// TwinCAT 3 PLC project PLC1
// ProgramVersion: 3.1.4026.27
// libraries:
//   Tc2_Standard, * (Beckhoff Automation GmbH)
//   Tc2_System, * (Beckhoff Automation GmbH)
//   Tc2_Utilities, * (Beckhoff Automation GmbH)
//   XPlanarApplication, * (Beckhoff Automation LLC)
// project tree:
//   DemoStep/ E_DemoStep.TcDUT, I_BothMovers.TcIO, I_Errorable.TcIO, I_SingleMover.TcIO, I_XplanarTable.TcIO, I_DemoStep.TcIO
//   DemoStep/Steps/ DetectXplanarMovers.TcPOU, LiftMove.TcPOU, SimpleDisableWithRotSwAndEstop.TcPOU, SimpleDisableWithPB.TcPOU, TiltMove.TcPOU, SpinMove.TcPOU, MoveAroundPerimeter.TcPOU, JoinAllClosestTracks.TcPOU, MoveAroundInSequence.TcPOU, OscillateRotateMove.TcPOU, RecoverMoveToAnyPos.TcPOU, FlyByMove.TcPOU, MoveToCenters.TcPOU, SameTrackMove.TcPOU, LeaveAllTracks.TcPOU, SimpleSort2Movers.TcPOU, SquareUpMovers.TcPOU, WaitForRotSw.TcPOU, InitStep.TcPOU, WaitForPB.TcPOU
//   DUTs/EStop/ E_EStop.TcDUT, ST_EstopIO.TcDUT, U_Estop.TcDUT
//   DUTs/ E_ButtonColors.TcDUT, E_UsbLicenseDongleSate.TcDUT, ST_Point.TcDUT (not stored)
//   DUTs/SelectorSwitch/ E_SelectorSwitchPos.TcDUT, ST_SelectorSwitchIO.TcDUT, U_SelectorSwitch.TcDUT
//   GVLs/ CoorPoint2Tile.TcGVL, Defaults.TcGVL
//   / PlcTask.TcTTO
//   POUs/ FB_PushButton.TcPOU, FB_ToggleButton.TcPOU, F_FindCorrectOpposingCornerPosition.TcPOU, F_FindOpposingRotationPosition.TcPOU, F_SetAllMoversMovement.TcPOU (not stored), F_SetAllMoversRotation.TcPOU (not stored), I_DemoSystem.TcIO, MAIN.TcPOU
// real-time tasks:
//   TASK PlcTask: cycle T#1ms, priority 20, ADS port 350
//   TASK Job Task: cycle default, priority 32
//   TASK XPlanar Task_3: cycle T#250us, priority 1, ADS port 351
//   TASK MC-Task (MET): cycle T#2ms, priority 2, ADS port 352
//   TASK MC-Task (MPT): cycle T#10ms, priority 3, ADS port 353
// I/O:
//   DEVICE XPlanar, AmsNetId 0.0.0.0.4.1
//     Term 1 (APS4322-7000) [APS4322-7000 Drive]
//       Term 2 (APS4322-5000) [APS4322-5000 Feedback]
//     Term 3 (APS4322-7000) [APS4322-7000 Drive]
//       Term 4 (APS4322-5000) [APS4322-5000 Feedback]
//   DEVICE IO (EtherCAT), AmsNetId 0.0.0.0.2.1
//     EtherCAT PS (PS2001-2410) [PS2001-2410-1001 Power supply (24V, 10A, 1-phase)]
//     IoLink PushButtons (EP6224-0002) [EP6224-0002 (IO Link Master)]
//       modules: Module 1 (DeviceState Inputs Device), Module 2 (DeviceState Inputs), Port1 (CANEO series10 Hygienic), Port2 (CANEO series10 Hygienic), Port3 (CANEO series10 Hygienic), Module 6 (empty), Module 7 (Digital Inputs)
//     DIO Box (RS and ESTOP) (EP2316-0003) [EP2316-0003 8 Ch. Dig. In, 10µs, 8Ch. Dig. Out 24V, 0,5A, Diagnostic, 10-Pole Plug Connector] (disabled)
//   DEVICE USB
//     Box 2 (C9900-L100 License-Key-USB-Stick)
// variable links:
//   PLC1/PLC1 Instance <-> IO (EtherCAT)
//     PlcTask Inputs/MAIN.IODeviceState <-> Inputs/DevState
//   PLC1/PLC1 Instance <-> USB/Box 2 (C9900-L100 License-Key-USB-Stick)
//     PlcTask Inputs/MAIN.LicUsbState <-> BoxInfo/BoxState
//   PLC1/PLC1 Instance <-> XPlanar
//     PlcTask Inputs/MAIN.XPlanarDeviceState <-> Inputs/DevState
//   PLC1/PLC1 Instance <-> XPlanar MC Project/Axes/Mover4220_1
//     PlcTask Inputs/MAIN.Mover1._Mover.MCTOPLC/ACT <-> McToPlc/ACT
//     PlcTask Inputs/MAIN.Mover1._Mover.MCTOPLC/COORDMODE <-> McToPlc/COORDMODE
//     PlcTask Inputs/MAIN.Mover1._Mover.MCTOPLC/SET <-> McToPlc/SET
//     PlcTask Inputs/MAIN.Mover1._Mover.MCTOPLC/SETONTRACK <-> McToPlc/SETONTRACK
//     PlcTask Inputs/MAIN.Mover1._Mover.MCTOPLC/STD <-> McToPlc/STD
//     PlcTask Outputs/MAIN.Mover1._Mover.PLCTOMC/STD <-> PlcToMc/STD
//   PLC1/PLC1 Instance <-> XPlanar MC Project/Axes/Mover4220_2
//     PlcTask Inputs/MAIN.Mover2._Mover.MCTOPLC/ACT <-> McToPlc/ACT
//     PlcTask Inputs/MAIN.Mover2._Mover.MCTOPLC/COORDMODE <-> McToPlc/COORDMODE
//     PlcTask Inputs/MAIN.Mover2._Mover.MCTOPLC/SET <-> McToPlc/SET
//     PlcTask Inputs/MAIN.Mover2._Mover.MCTOPLC/SETONTRACK <-> McToPlc/SETONTRACK
//     PlcTask Inputs/MAIN.Mover2._Mover.MCTOPLC/STD <-> McToPlc/STD
//     PlcTask Outputs/MAIN.Mover2._Mover.PLCTOMC/STD <-> PlcToMc/STD
//   PLC1/PLC1 Instance <-> XPlanar MC Project/Groups/Environment
//     PlcTask Inputs/XPlanar.Environment.MCTOPLC_STD <-> McToPlc/STD
//   PLC1/PLC1 Instance <-> XPlanar MC Project/Groups/Track_Fig8
//     PlcTask Inputs/MAIN.Track1._Track.MCTOPLC_STD <-> McToPlc/STD
//   PLC1/PLC1 Instance <-> XPlanar MC Project/Groups/XPlanar
//     PlcTask Inputs/XPlanar.Group.MCTOPLC_STD <-> McToPlc/STD
//   TcCOM Objects/XPlanar <-> XPlanar/Term 1 (APS4322-7000)
//     Part1/APS4322_P1_2/Data Pointer/DCurrentSetPoints[0] <-> APS Outputs/Current D 0X0
//     Part1/APS4322_P1_2/Data Pointer/DCurrentSetPoints[12] <-> APS Outputs/Current D 2X0
//     Part1/APS4322_P1_2/Data Pointer/DCurrentSetPoints[13] <-> APS Outputs/Current D 2X1
//     Part1/APS4322_P1_2/Data Pointer/DCurrentSetPoints[14] <-> APS Outputs/Current D 2X2
//     Part1/APS4322_P1_2/Data Pointer/DCurrentSetPoints[18] <-> APS Outputs/Current D 3X0
//     Part1/APS4322_P1_2/Data Pointer/DCurrentSetPoints[19] <-> APS Outputs/Current D 3X1
//     Part1/APS4322_P1_2/Data Pointer/DCurrentSetPoints[1] <-> APS Outputs/Current D 0X1
//     Part1/APS4322_P1_2/Data Pointer/DCurrentSetPoints[20] <-> APS Outputs/Current D 3X2
//     Part1/APS4322_P1_2/Data Pointer/DCurrentSetPoints[2] <-> APS Outputs/Current D 0X2
//     Part1/APS4322_P1_2/Data Pointer/DCurrentSetPoints[6] <-> APS Outputs/Current D 1X0
//     Part1/APS4322_P1_2/Data Pointer/DCurrentSetPoints[7] <-> APS Outputs/Current D 1X1
//     Part1/APS4322_P1_2/Data Pointer/DCurrentSetPoints[8] <-> APS Outputs/Current D 1X2
//     Part1/APS4322_P1_2/Data Pointer/DCurrentSetPoints[10] <-> APS Outputs/Current D 1Y1
//     Part1/APS4322_P1_2/Data Pointer/DCurrentSetPoints[11] <-> APS Outputs/Current D 1Y2
//     Part1/APS4322_P1_2/Data Pointer/DCurrentSetPoints[15] <-> APS Outputs/Current D 2Y0
//     Part1/APS4322_P1_2/Data Pointer/DCurrentSetPoints[16] <-> APS Outputs/Current D 2Y1
//     Part1/APS4322_P1_2/Data Pointer/DCurrentSetPoints[17] <-> APS Outputs/Current D 2Y2
//     Part1/APS4322_P1_2/Data Pointer/DCurrentSetPoints[21] <-> APS Outputs/Current D 3Y0
//     Part1/APS4322_P1_2/Data Pointer/DCurrentSetPoints[22] <-> APS Outputs/Current D 3Y1
//     Part1/APS4322_P1_2/Data Pointer/DCurrentSetPoints[23] <-> APS Outputs/Current D 3Y2
//     Part1/APS4322_P1_2/Data Pointer/DCurrentSetPoints[3] <-> APS Outputs/Current D 0Y0
//     Part1/APS4322_P1_2/Data Pointer/DCurrentSetPoints[4] <-> APS Outputs/Current D 0Y1
//     Part1/APS4322_P1_2/Data Pointer/DCurrentSetPoints[5] <-> APS Outputs/Current D 0Y2
//     Part1/APS4322_P1_2/Data Pointer/DCurrentSetPoints[9] <-> APS Outputs/Current D 1Y0
//     Part1/APS4322_P1_2/Data Pointer/DcLinkVoltage <-> APS Diagdata/DC Link Voltage
//     Part1/APS4322_P1_2/Data Pointer/MoverCommControlWord <-> APS Comm Outputs/CommControlWord
//     Part1/APS4322_P1_2/Data Pointer/MoverCommDataIn[{0..3}] <-> APS Comm Inputs/Data {1..4}  (4 links)
//     Part1/APS4322_P1_2/Data Pointer/MoverCommDataOut <-> APS Comm Outputs/Data 1
//     Part1/APS4322_P1_2/Data Pointer/MoverCommStatusWord <-> APS Comm Inputs/CommStatusWord
//     Part1/APS4322_P1_2/Data Pointer/PhiSetPoints[0] <-> APS Outputs/PhiE 0X0
//     Part1/APS4322_P1_2/Data Pointer/PhiSetPoints[12] <-> APS Outputs/PhiE 2X0
//     Part1/APS4322_P1_2/Data Pointer/PhiSetPoints[13] <-> APS Outputs/PhiE 2X1
//     Part1/APS4322_P1_2/Data Pointer/PhiSetPoints[14] <-> APS Outputs/PhiE 2X2
//     Part1/APS4322_P1_2/Data Pointer/PhiSetPoints[18] <-> APS Outputs/PhiE 3X0
//     Part1/APS4322_P1_2/Data Pointer/PhiSetPoints[19] <-> APS Outputs/PhiE 3X1
//     Part1/APS4322_P1_2/Data Pointer/PhiSetPoints[1] <-> APS Outputs/PhiE 0X1
//     Part1/APS4322_P1_2/Data Pointer/PhiSetPoints[20] <-> APS Outputs/PhiE 3X2
//     Part1/APS4322_P1_2/Data Pointer/PhiSetPoints[2] <-> APS Outputs/PhiE 0X2
//     Part1/APS4322_P1_2/Data Pointer/PhiSetPoints[6] <-> APS Outputs/PhiE 1X0
//     Part1/APS4322_P1_2/Data Pointer/PhiSetPoints[7] <-> APS Outputs/PhiE 1X1
//     Part1/APS4322_P1_2/Data Pointer/PhiSetPoints[8] <-> APS Outputs/PhiE 1X2
//     Part1/APS4322_P1_2/Data Pointer/PhiSetPoints[10] <-> APS Outputs/PhiE 1Y1
//     Part1/APS4322_P1_2/Data Pointer/PhiSetPoints[11] <-> APS Outputs/PhiE 1Y2
//     Part1/APS4322_P1_2/Data Pointer/PhiSetPoints[15] <-> APS Outputs/PhiE 2Y0
//     Part1/APS4322_P1_2/Data Pointer/PhiSetPoints[16] <-> APS Outputs/PhiE 2Y1
//     Part1/APS4322_P1_2/Data Pointer/PhiSetPoints[17] <-> APS Outputs/PhiE 2Y2
//     Part1/APS4322_P1_2/Data Pointer/PhiSetPoints[21] <-> APS Outputs/PhiE 3Y0
//     Part1/APS4322_P1_2/Data Pointer/PhiSetPoints[22] <-> APS Outputs/PhiE 3Y1
//     Part1/APS4322_P1_2/Data Pointer/PhiSetPoints[23] <-> APS Outputs/PhiE 3Y2
//     Part1/APS4322_P1_2/Data Pointer/PhiSetPoints[3] <-> APS Outputs/PhiE 0Y0
//     Part1/APS4322_P1_2/Data Pointer/PhiSetPoints[4] <-> APS Outputs/PhiE 0Y1
//     Part1/APS4322_P1_2/Data Pointer/PhiSetPoints[5] <-> APS Outputs/PhiE 0Y2
//     Part1/APS4322_P1_2/Data Pointer/PhiSetPoints[9] <-> APS Outputs/PhiE 1Y0
//     Part1/APS4322_P1_2/Data Pointer/PowerSupplyCurrent <-> APS Diagdata/Power supply current
//     Part1/APS4322_P1_2/Data Pointer/PowerUnitControlWord <-> APS Outputs/ControlWord
//     Part1/APS4322_P1_2/Data Pointer/PowerUnitStatusWord <-> APS Inputs/StatusWord
//     Part1/APS4322_P1_2/Data Pointer/QCurrentSetPoints[0] <-> APS Outputs/Current Q 0X0
//     Part1/APS4322_P1_2/Data Pointer/QCurrentSetPoints[12] <-> APS Outputs/Current Q 2X0
//     Part1/APS4322_P1_2/Data Pointer/QCurrentSetPoints[13] <-> APS Outputs/Current Q 2X1
//     Part1/APS4322_P1_2/Data Pointer/QCurrentSetPoints[14] <-> APS Outputs/Current Q 2X2
//     Part1/APS4322_P1_2/Data Pointer/QCurrentSetPoints[18] <-> APS Outputs/Current Q 3X0
//     Part1/APS4322_P1_2/Data Pointer/QCurrentSetPoints[19] <-> APS Outputs/Current Q 3X1
//     Part1/APS4322_P1_2/Data Pointer/QCurrentSetPoints[1] <-> APS Outputs/Current Q 0X1
//     Part1/APS4322_P1_2/Data Pointer/QCurrentSetPoints[20] <-> APS Outputs/Current Q 3X2
//     Part1/APS4322_P1_2/Data Pointer/QCurrentSetPoints[2] <-> APS Outputs/Current Q 0X2
//     Part1/APS4322_P1_2/Data Pointer/QCurrentSetPoints[6] <-> APS Outputs/Current Q 1X0
//     Part1/APS4322_P1_2/Data Pointer/QCurrentSetPoints[7] <-> APS Outputs/Current Q 1X1
//     Part1/APS4322_P1_2/Data Pointer/QCurrentSetPoints[8] <-> APS Outputs/Current Q 1X2
//     Part1/APS4322_P1_2/Data Pointer/QCurrentSetPoints[10] <-> APS Outputs/Current Q 1Y1
//     Part1/APS4322_P1_2/Data Pointer/QCurrentSetPoints[11] <-> APS Outputs/Current Q 1Y2
//     Part1/APS4322_P1_2/Data Pointer/QCurrentSetPoints[15] <-> APS Outputs/Current Q 2Y0
//     Part1/APS4322_P1_2/Data Pointer/QCurrentSetPoints[16] <-> APS Outputs/Current Q 2Y1
//     Part1/APS4322_P1_2/Data Pointer/QCurrentSetPoints[17] <-> APS Outputs/Current Q 2Y2
//     Part1/APS4322_P1_2/Data Pointer/QCurrentSetPoints[21] <-> APS Outputs/Current Q 3Y0
//     Part1/APS4322_P1_2/Data Pointer/QCurrentSetPoints[22] <-> APS Outputs/Current Q 3Y1
//     Part1/APS4322_P1_2/Data Pointer/QCurrentSetPoints[23] <-> APS Outputs/Current Q 3Y2
//     Part1/APS4322_P1_2/Data Pointer/QCurrentSetPoints[3] <-> APS Outputs/Current Q 0Y0
//     Part1/APS4322_P1_2/Data Pointer/QCurrentSetPoints[4] <-> APS Outputs/Current Q 0Y1
//     Part1/APS4322_P1_2/Data Pointer/QCurrentSetPoints[5] <-> APS Outputs/Current Q 0Y2
//     Part1/APS4322_P1_2/Data Pointer/QCurrentSetPoints[9] <-> APS Outputs/Current Q 1Y0
//   TcCOM Objects/XPlanar <-> XPlanar/Term 1 (APS4322-7000)/Term 2 (APS4322-5000)
//     Part1/APS4322_P1_2/Data Pointer/FeedbackStatus <-> FB Inputs/Status
//     Part1/APS4322_P1_2/Data Pointer/HallSensorFieldsXYZ[{0..12 step 3}] <-> FB Inputs/A{0..8 step 2} X-Field  (5 links)
//     Part1/APS4322_P1_2/Data Pointer/HallSensorFieldsXYZ[{91..103 step 3}] <-> FB Inputs/G{0..8 step 2} Y-Field  (5 links)
//     Part1/APS4322_P1_2/Data Pointer/HallSensorFieldsXYZ[{92..104 step 3}] <-> FB Inputs/G{0..8 step 2} Z-Field  (5 links)
//     Part1/APS4322_P1_2/Data Pointer/HallSensorFieldsXYZ[{90..102 step 3}] <-> FB Inputs/G{0..8 step 2} X-Field  (5 links)
//     Part1/APS4322_P1_2/Data Pointer/HallSensorFieldsXYZ[{105..117 step 3}] <-> FB Inputs/H{1..9 step 2} X-Field  (5 links)
//     Part1/APS4322_P1_2/Data Pointer/HallSensorFieldsXYZ[{106..118 step 3}] <-> FB Inputs/H{1..9 step 2} Y-Field  (5 links)
//     Part1/APS4322_P1_2/Data Pointer/HallSensorFieldsXYZ[{107..119 step 3}] <-> FB Inputs/H{1..9 step 2} Z-Field  (5 links)
//     Part1/APS4322_P1_2/Data Pointer/HallSensorFieldsXYZ[{1..13 step 3}] <-> FB Inputs/A{0..8 step 2} Y-Field  (5 links)
//     Part1/APS4322_P1_2/Data Pointer/HallSensorFieldsXYZ[{2..14 step 3}] <-> FB Inputs/A{0..8 step 2} Z-Field  (5 links)
//     Part1/APS4322_P1_2/Data Pointer/HallSensorFieldsXYZ[{120..132 step 3}] <-> FB Inputs/I{0..8 step 2} X-Field  (5 links)
//     Part1/APS4322_P1_2/Data Pointer/HallSensorFieldsXYZ[{121..133 step 3}] <-> FB Inputs/I{0..8 step 2} Y-Field  (5 links)
//     Part1/APS4322_P1_2/Data Pointer/HallSensorFieldsXYZ[{122..134 step 3}] <-> FB Inputs/I{0..8 step 2} Z-Field  (5 links)
//     Part1/APS4322_P1_2/Data Pointer/HallSensorFieldsXYZ[{135..147 step 3}] <-> FB Inputs/J{1..9 step 2} X-Field  (5 links)
//     Part1/APS4322_P1_2/Data Pointer/HallSensorFieldsXYZ[{136..148 step 3}] <-> FB Inputs/J{1..9 step 2} Y-Field  (5 links)
//     Part1/APS4322_P1_2/Data Pointer/HallSensorFieldsXYZ[{137..149 step 3}] <-> FB Inputs/J{1..9 step 2} Z-Field  (5 links)
//     Part1/APS4322_P1_2/Data Pointer/HallSensorFieldsXYZ[{15..27 step 3}] <-> FB Inputs/B{1..9 step 2} X-Field  (5 links)
//     Part1/APS4322_P1_2/Data Pointer/HallSensorFieldsXYZ[{16..28 step 3}] <-> FB Inputs/B{1..9 step 2} Y-Field  (5 links)
//     Part1/APS4322_P1_2/Data Pointer/HallSensorFieldsXYZ[{17..29 step 3}] <-> FB Inputs/B{1..9 step 2} Z-Field  (5 links)
//     Part1/APS4322_P1_2/Data Pointer/HallSensorFieldsXYZ[{30..42 step 3}] <-> FB Inputs/C{0..8 step 2} X-Field  (5 links)
//     Part1/APS4322_P1_2/Data Pointer/HallSensorFieldsXYZ[{31..43 step 3}] <-> FB Inputs/C{0..8 step 2} Y-Field  (5 links)
//     Part1/APS4322_P1_2/Data Pointer/HallSensorFieldsXYZ[{32..44 step 3}] <-> FB Inputs/C{0..8 step 2} Z-Field  (5 links)
//     Part1/APS4322_P1_2/Data Pointer/HallSensorFieldsXYZ[{45..57 step 3}] <-> FB Inputs/D{1..9 step 2} X-Field  (5 links)
//     Part1/APS4322_P1_2/Data Pointer/HallSensorFieldsXYZ[{46..58 step 3}] <-> FB Inputs/D{1..9 step 2} Y-Field  (5 links)
//     Part1/APS4322_P1_2/Data Pointer/HallSensorFieldsXYZ[{47..59 step 3}] <-> FB Inputs/D{1..9 step 2} Z-Field  (5 links)
//     Part1/APS4322_P1_2/Data Pointer/HallSensorFieldsXYZ[{60..72 step 3}] <-> FB Inputs/E{0..8 step 2} X-Field  (5 links)
//     Part1/APS4322_P1_2/Data Pointer/HallSensorFieldsXYZ[{61..73 step 3}] <-> FB Inputs/E{0..8 step 2} Y-Field  (5 links)
//     Part1/APS4322_P1_2/Data Pointer/HallSensorFieldsXYZ[{62..74 step 3}] <-> FB Inputs/E{0..8 step 2} Z-Field  (5 links)
//     Part1/APS4322_P1_2/Data Pointer/HallSensorFieldsXYZ[{75..87 step 3}] <-> FB Inputs/F{1..9 step 2} X-Field  (5 links)
//     Part1/APS4322_P1_2/Data Pointer/HallSensorFieldsXYZ[{76..88 step 3}] <-> FB Inputs/F{1..9 step 2} Y-Field  (5 links)
//     Part1/APS4322_P1_2/Data Pointer/HallSensorFieldsXYZ[{77..89 step 3}] <-> FB Inputs/F{1..9 step 2} Z-Field  (5 links)
//   TcCOM Objects/XPlanar <-> XPlanar/Term 3 (APS4322-7000)
//     Part1/APS4322_P1_1/Data Pointer/DCurrentSetPoints[0] <-> APS Outputs/Current D 0X0
//     Part1/APS4322_P1_1/Data Pointer/DCurrentSetPoints[12] <-> APS Outputs/Current D 2X0
//     Part1/APS4322_P1_1/Data Pointer/DCurrentSetPoints[13] <-> APS Outputs/Current D 2X1
//     Part1/APS4322_P1_1/Data Pointer/DCurrentSetPoints[14] <-> APS Outputs/Current D 2X2
//     Part1/APS4322_P1_1/Data Pointer/DCurrentSetPoints[18] <-> APS Outputs/Current D 3X0
//     Part1/APS4322_P1_1/Data Pointer/DCurrentSetPoints[19] <-> APS Outputs/Current D 3X1
//     Part1/APS4322_P1_1/Data Pointer/DCurrentSetPoints[1] <-> APS Outputs/Current D 0X1
//     Part1/APS4322_P1_1/Data Pointer/DCurrentSetPoints[20] <-> APS Outputs/Current D 3X2
//     Part1/APS4322_P1_1/Data Pointer/DCurrentSetPoints[2] <-> APS Outputs/Current D 0X2
//     Part1/APS4322_P1_1/Data Pointer/DCurrentSetPoints[6] <-> APS Outputs/Current D 1X0
//     Part1/APS4322_P1_1/Data Pointer/DCurrentSetPoints[7] <-> APS Outputs/Current D 1X1
//     Part1/APS4322_P1_1/Data Pointer/DCurrentSetPoints[8] <-> APS Outputs/Current D 1X2
//     Part1/APS4322_P1_1/Data Pointer/DCurrentSetPoints[10] <-> APS Outputs/Current D 1Y1
//     Part1/APS4322_P1_1/Data Pointer/DCurrentSetPoints[11] <-> APS Outputs/Current D 1Y2
//     Part1/APS4322_P1_1/Data Pointer/DCurrentSetPoints[15] <-> APS Outputs/Current D 2Y0
//     Part1/APS4322_P1_1/Data Pointer/DCurrentSetPoints[16] <-> APS Outputs/Current D 2Y1
//     Part1/APS4322_P1_1/Data Pointer/DCurrentSetPoints[17] <-> APS Outputs/Current D 2Y2
//     Part1/APS4322_P1_1/Data Pointer/DCurrentSetPoints[21] <-> APS Outputs/Current D 3Y0
//     Part1/APS4322_P1_1/Data Pointer/DCurrentSetPoints[22] <-> APS Outputs/Current D 3Y1
//     Part1/APS4322_P1_1/Data Pointer/DCurrentSetPoints[23] <-> APS Outputs/Current D 3Y2
//     Part1/APS4322_P1_1/Data Pointer/DCurrentSetPoints[3] <-> APS Outputs/Current D 0Y0
//     Part1/APS4322_P1_1/Data Pointer/DCurrentSetPoints[4] <-> APS Outputs/Current D 0Y1
//     Part1/APS4322_P1_1/Data Pointer/DCurrentSetPoints[5] <-> APS Outputs/Current D 0Y2
//     Part1/APS4322_P1_1/Data Pointer/DCurrentSetPoints[9] <-> APS Outputs/Current D 1Y0
//     Part1/APS4322_P1_1/Data Pointer/DcLinkVoltage <-> APS Diagdata/DC Link Voltage
//     Part1/APS4322_P1_1/Data Pointer/MoverCommControlWord <-> APS Comm Outputs/CommControlWord
//     Part1/APS4322_P1_1/Data Pointer/MoverCommDataIn[{0..3}] <-> APS Comm Inputs/Data {1..4}  (4 links)
//     Part1/APS4322_P1_1/Data Pointer/MoverCommDataOut <-> APS Comm Outputs/Data 1
//     Part1/APS4322_P1_1/Data Pointer/MoverCommStatusWord <-> APS Comm Inputs/CommStatusWord
//     Part1/APS4322_P1_1/Data Pointer/PhiSetPoints[0] <-> APS Outputs/PhiE 0X0
//     Part1/APS4322_P1_1/Data Pointer/PhiSetPoints[12] <-> APS Outputs/PhiE 2X0
//     Part1/APS4322_P1_1/Data Pointer/PhiSetPoints[13] <-> APS Outputs/PhiE 2X1
//     Part1/APS4322_P1_1/Data Pointer/PhiSetPoints[14] <-> APS Outputs/PhiE 2X2
//     Part1/APS4322_P1_1/Data Pointer/PhiSetPoints[18] <-> APS Outputs/PhiE 3X0
//     Part1/APS4322_P1_1/Data Pointer/PhiSetPoints[19] <-> APS Outputs/PhiE 3X1
//     Part1/APS4322_P1_1/Data Pointer/PhiSetPoints[1] <-> APS Outputs/PhiE 0X1
//     Part1/APS4322_P1_1/Data Pointer/PhiSetPoints[20] <-> APS Outputs/PhiE 3X2
//     Part1/APS4322_P1_1/Data Pointer/PhiSetPoints[2] <-> APS Outputs/PhiE 0X2
//     Part1/APS4322_P1_1/Data Pointer/PhiSetPoints[6] <-> APS Outputs/PhiE 1X0
//     Part1/APS4322_P1_1/Data Pointer/PhiSetPoints[7] <-> APS Outputs/PhiE 1X1
//     Part1/APS4322_P1_1/Data Pointer/PhiSetPoints[8] <-> APS Outputs/PhiE 1X2
//     Part1/APS4322_P1_1/Data Pointer/PhiSetPoints[10] <-> APS Outputs/PhiE 1Y1
//     Part1/APS4322_P1_1/Data Pointer/PhiSetPoints[11] <-> APS Outputs/PhiE 1Y2
//     Part1/APS4322_P1_1/Data Pointer/PhiSetPoints[15] <-> APS Outputs/PhiE 2Y0
//     Part1/APS4322_P1_1/Data Pointer/PhiSetPoints[16] <-> APS Outputs/PhiE 2Y1
//     Part1/APS4322_P1_1/Data Pointer/PhiSetPoints[17] <-> APS Outputs/PhiE 2Y2
//     Part1/APS4322_P1_1/Data Pointer/PhiSetPoints[21] <-> APS Outputs/PhiE 3Y0
//     Part1/APS4322_P1_1/Data Pointer/PhiSetPoints[22] <-> APS Outputs/PhiE 3Y1
//     Part1/APS4322_P1_1/Data Pointer/PhiSetPoints[23] <-> APS Outputs/PhiE 3Y2
//     Part1/APS4322_P1_1/Data Pointer/PhiSetPoints[3] <-> APS Outputs/PhiE 0Y0
//     Part1/APS4322_P1_1/Data Pointer/PhiSetPoints[4] <-> APS Outputs/PhiE 0Y1
//     Part1/APS4322_P1_1/Data Pointer/PhiSetPoints[5] <-> APS Outputs/PhiE 0Y2
//     Part1/APS4322_P1_1/Data Pointer/PhiSetPoints[9] <-> APS Outputs/PhiE 1Y0
//     Part1/APS4322_P1_1/Data Pointer/PowerSupplyCurrent <-> APS Diagdata/Power supply current
//     Part1/APS4322_P1_1/Data Pointer/PowerUnitControlWord <-> APS Outputs/ControlWord
//     Part1/APS4322_P1_1/Data Pointer/PowerUnitStatusWord <-> APS Inputs/StatusWord
//     Part1/APS4322_P1_1/Data Pointer/QCurrentSetPoints[0] <-> APS Outputs/Current Q 0X0
//     Part1/APS4322_P1_1/Data Pointer/QCurrentSetPoints[12] <-> APS Outputs/Current Q 2X0
//     Part1/APS4322_P1_1/Data Pointer/QCurrentSetPoints[13] <-> APS Outputs/Current Q 2X1
//     Part1/APS4322_P1_1/Data Pointer/QCurrentSetPoints[14] <-> APS Outputs/Current Q 2X2
//     Part1/APS4322_P1_1/Data Pointer/QCurrentSetPoints[18] <-> APS Outputs/Current Q 3X0
//     Part1/APS4322_P1_1/Data Pointer/QCurrentSetPoints[19] <-> APS Outputs/Current Q 3X1
//     Part1/APS4322_P1_1/Data Pointer/QCurrentSetPoints[1] <-> APS Outputs/Current Q 0X1
//     Part1/APS4322_P1_1/Data Pointer/QCurrentSetPoints[20] <-> APS Outputs/Current Q 3X2
//     Part1/APS4322_P1_1/Data Pointer/QCurrentSetPoints[2] <-> APS Outputs/Current Q 0X2
//     Part1/APS4322_P1_1/Data Pointer/QCurrentSetPoints[6] <-> APS Outputs/Current Q 1X0
//     Part1/APS4322_P1_1/Data Pointer/QCurrentSetPoints[7] <-> APS Outputs/Current Q 1X1
//     Part1/APS4322_P1_1/Data Pointer/QCurrentSetPoints[8] <-> APS Outputs/Current Q 1X2
//     Part1/APS4322_P1_1/Data Pointer/QCurrentSetPoints[10] <-> APS Outputs/Current Q 1Y1
//     Part1/APS4322_P1_1/Data Pointer/QCurrentSetPoints[11] <-> APS Outputs/Current Q 1Y2
//     Part1/APS4322_P1_1/Data Pointer/QCurrentSetPoints[15] <-> APS Outputs/Current Q 2Y0
//     Part1/APS4322_P1_1/Data Pointer/QCurrentSetPoints[16] <-> APS Outputs/Current Q 2Y1
//     Part1/APS4322_P1_1/Data Pointer/QCurrentSetPoints[17] <-> APS Outputs/Current Q 2Y2
//     Part1/APS4322_P1_1/Data Pointer/QCurrentSetPoints[21] <-> APS Outputs/Current Q 3Y0
//     Part1/APS4322_P1_1/Data Pointer/QCurrentSetPoints[22] <-> APS Outputs/Current Q 3Y1
//     Part1/APS4322_P1_1/Data Pointer/QCurrentSetPoints[23] <-> APS Outputs/Current Q 3Y2
//     Part1/APS4322_P1_1/Data Pointer/QCurrentSetPoints[3] <-> APS Outputs/Current Q 0Y0
//     Part1/APS4322_P1_1/Data Pointer/QCurrentSetPoints[4] <-> APS Outputs/Current Q 0Y1
//     Part1/APS4322_P1_1/Data Pointer/QCurrentSetPoints[5] <-> APS Outputs/Current Q 0Y2
//     Part1/APS4322_P1_1/Data Pointer/QCurrentSetPoints[9] <-> APS Outputs/Current Q 1Y0
//   TcCOM Objects/XPlanar <-> XPlanar/Term 3 (APS4322-7000)/Term 4 (APS4322-5000)
//     Part1/APS4322_P1_1/Data Pointer/FeedbackStatus <-> FB Inputs/Status
//     Part1/APS4322_P1_1/Data Pointer/HallSensorFieldsXYZ[{0..12 step 3}] <-> FB Inputs/A{0..8 step 2} X-Field  (5 links)
//     Part1/APS4322_P1_1/Data Pointer/HallSensorFieldsXYZ[{91..103 step 3}] <-> FB Inputs/G{0..8 step 2} Y-Field  (5 links)
//     Part1/APS4322_P1_1/Data Pointer/HallSensorFieldsXYZ[{92..104 step 3}] <-> FB Inputs/G{0..8 step 2} Z-Field  (5 links)
//     Part1/APS4322_P1_1/Data Pointer/HallSensorFieldsXYZ[{90..102 step 3}] <-> FB Inputs/G{0..8 step 2} X-Field  (5 links)
//     Part1/APS4322_P1_1/Data Pointer/HallSensorFieldsXYZ[{105..117 step 3}] <-> FB Inputs/H{1..9 step 2} X-Field  (5 links)
//     Part1/APS4322_P1_1/Data Pointer/HallSensorFieldsXYZ[{106..118 step 3}] <-> FB Inputs/H{1..9 step 2} Y-Field  (5 links)
//     Part1/APS4322_P1_1/Data Pointer/HallSensorFieldsXYZ[{107..119 step 3}] <-> FB Inputs/H{1..9 step 2} Z-Field  (5 links)
//     Part1/APS4322_P1_1/Data Pointer/HallSensorFieldsXYZ[{1..13 step 3}] <-> FB Inputs/A{0..8 step 2} Y-Field  (5 links)
//     Part1/APS4322_P1_1/Data Pointer/HallSensorFieldsXYZ[{2..14 step 3}] <-> FB Inputs/A{0..8 step 2} Z-Field  (5 links)
//     Part1/APS4322_P1_1/Data Pointer/HallSensorFieldsXYZ[{120..132 step 3}] <-> FB Inputs/I{0..8 step 2} X-Field  (5 links)
//     Part1/APS4322_P1_1/Data Pointer/HallSensorFieldsXYZ[{121..133 step 3}] <-> FB Inputs/I{0..8 step 2} Y-Field  (5 links)
//     Part1/APS4322_P1_1/Data Pointer/HallSensorFieldsXYZ[{122..134 step 3}] <-> FB Inputs/I{0..8 step 2} Z-Field  (5 links)
//     Part1/APS4322_P1_1/Data Pointer/HallSensorFieldsXYZ[{135..147 step 3}] <-> FB Inputs/J{1..9 step 2} X-Field  (5 links)
//     Part1/APS4322_P1_1/Data Pointer/HallSensorFieldsXYZ[{136..148 step 3}] <-> FB Inputs/J{1..9 step 2} Y-Field  (5 links)
//     Part1/APS4322_P1_1/Data Pointer/HallSensorFieldsXYZ[{137..149 step 3}] <-> FB Inputs/J{1..9 step 2} Z-Field  (5 links)
//     Part1/APS4322_P1_1/Data Pointer/HallSensorFieldsXYZ[{15..27 step 3}] <-> FB Inputs/B{1..9 step 2} X-Field  (5 links)
//     Part1/APS4322_P1_1/Data Pointer/HallSensorFieldsXYZ[{16..28 step 3}] <-> FB Inputs/B{1..9 step 2} Y-Field  (5 links)
//     Part1/APS4322_P1_1/Data Pointer/HallSensorFieldsXYZ[{17..29 step 3}] <-> FB Inputs/B{1..9 step 2} Z-Field  (5 links)
//     Part1/APS4322_P1_1/Data Pointer/HallSensorFieldsXYZ[{30..42 step 3}] <-> FB Inputs/C{0..8 step 2} X-Field  (5 links)
//     Part1/APS4322_P1_1/Data Pointer/HallSensorFieldsXYZ[{31..43 step 3}] <-> FB Inputs/C{0..8 step 2} Y-Field  (5 links)
//     Part1/APS4322_P1_1/Data Pointer/HallSensorFieldsXYZ[{32..44 step 3}] <-> FB Inputs/C{0..8 step 2} Z-Field  (5 links)
//     Part1/APS4322_P1_1/Data Pointer/HallSensorFieldsXYZ[{45..57 step 3}] <-> FB Inputs/D{1..9 step 2} X-Field  (5 links)
//     Part1/APS4322_P1_1/Data Pointer/HallSensorFieldsXYZ[{46..58 step 3}] <-> FB Inputs/D{1..9 step 2} Y-Field  (5 links)
//     Part1/APS4322_P1_1/Data Pointer/HallSensorFieldsXYZ[{47..59 step 3}] <-> FB Inputs/D{1..9 step 2} Z-Field  (5 links)
//     Part1/APS4322_P1_1/Data Pointer/HallSensorFieldsXYZ[{60..72 step 3}] <-> FB Inputs/E{0..8 step 2} X-Field  (5 links)
//     Part1/APS4322_P1_1/Data Pointer/HallSensorFieldsXYZ[{61..73 step 3}] <-> FB Inputs/E{0..8 step 2} Y-Field  (5 links)
//     Part1/APS4322_P1_1/Data Pointer/HallSensorFieldsXYZ[{62..74 step 3}] <-> FB Inputs/E{0..8 step 2} Z-Field  (5 links)
//     Part1/APS4322_P1_1/Data Pointer/HallSensorFieldsXYZ[{75..87 step 3}] <-> FB Inputs/F{1..9 step 2} X-Field  (5 links)
//     Part1/APS4322_P1_1/Data Pointer/HallSensorFieldsXYZ[{76..88 step 3}] <-> FB Inputs/F{1..9 step 2} Y-Field  (5 links)
//     Part1/APS4322_P1_1/Data Pointer/HallSensorFieldsXYZ[{77..89 step 3}] <-> FB Inputs/F{1..9 step 2} Z-Field  (5 links)
//   TcCOM Objects/XPlanar <-> XPlanar MC Project/Axes/Mover4220_1
//     Mover4220_1/InputsFromNC3/NC3ToHW <-> McToIo/STD
//     Mover4220_1/OutputsToNC3/HWToNC3 <-> IoToMc/STD
//   TcCOM Objects/XPlanar <-> XPlanar MC Project/Axes/Mover4220_2
//     Mover4220_2/InputsFromNC3/NC3ToHW <-> McToIo/STD
//     Mover4220_2/OutputsToNC3/HWToNC3 <-> IoToMc/STD
//   __THIS__ <-> PLC1/PLC1 Instance
//     Port1 (CANEO series10 Hygienic)/IO-Link Port1_in/Actuation Count <-> PlcTask Inputs/MAIN.START_Button.actuation_count
//     Port1 (CANEO series10 Hygienic)/IO-Link Port1_in/Actuation Flag <-> PlcTask Inputs/MAIN.START_Button.actuation_flag
//     Port1 (CANEO series10 Hygienic)/IO-Link Port1_in/Actuation Strength <-> PlcTask Inputs/MAIN.START_Button.actuation_strength
//     Port1 (CANEO series10 Hygienic)/IO-Link Port1_in/Surrounding Brightness <-> PlcTask Inputs/MAIN.START_Button.surrounding_brightness
//     Port1 (CANEO series10 Hygienic)/IO-Link Port1_out/Active LEDs <-> PlcTask Outputs/MAIN.START_Button.active_leds
//     Port1 (CANEO series10 Hygienic)/IO-Link Port1_out/Effect Frequency <-> PlcTask Outputs/MAIN.START_Button.effect_frequency
//     Port1 (CANEO series10 Hygienic)/IO-Link Port1_out/LED Brightness <-> PlcTask Outputs/MAIN.START_Button.led_brightness
//     Port1 (CANEO series10 Hygienic)/IO-Link Port1_out/LED Color B <-> PlcTask Outputs/MAIN.START_Button.led_blue
//     Port1 (CANEO series10 Hygienic)/IO-Link Port1_out/LED Color G <-> PlcTask Outputs/MAIN.START_Button.led_green
//     Port1 (CANEO series10 Hygienic)/IO-Link Port1_out/LED Color R <-> PlcTask Outputs/MAIN.START_Button.led_red
//     Port1 (CANEO series10 Hygienic)/IO-Link Port1_out/LED Effect <-> PlcTask Outputs/MAIN.START_Button.led_effect
//     Port2 (CANEO series10 Hygienic)/IO-Link Port2_in/Actuation Count <-> PlcTask Inputs/MAIN.DISABLE_Button.actuation_count
//     Port2 (CANEO series10 Hygienic)/IO-Link Port2_in/Actuation Flag <-> PlcTask Inputs/MAIN.DISABLE_Button.actuation_flag
//     Port2 (CANEO series10 Hygienic)/IO-Link Port2_in/Actuation Strength <-> PlcTask Inputs/MAIN.DISABLE_Button.actuation_strength
//     Port2 (CANEO series10 Hygienic)/IO-Link Port2_in/Surrounding Brightness <-> PlcTask Inputs/MAIN.DISABLE_Button.surrounding_brightness
//     Port2 (CANEO series10 Hygienic)/IO-Link Port2_out/Active LEDs <-> PlcTask Outputs/MAIN.DISABLE_Button.active_leds
//     Port2 (CANEO series10 Hygienic)/IO-Link Port2_out/Effect Frequency <-> PlcTask Outputs/MAIN.DISABLE_Button.effect_frequency
//     Port2 (CANEO series10 Hygienic)/IO-Link Port2_out/LED Brightness <-> PlcTask Outputs/MAIN.DISABLE_Button.led_brightness
//     Port2 (CANEO series10 Hygienic)/IO-Link Port2_out/LED Color B <-> PlcTask Outputs/MAIN.DISABLE_Button.led_blue
//     Port2 (CANEO series10 Hygienic)/IO-Link Port2_out/LED Color G <-> PlcTask Outputs/MAIN.DISABLE_Button.led_green
//     Port2 (CANEO series10 Hygienic)/IO-Link Port2_out/LED Color R <-> PlcTask Outputs/MAIN.DISABLE_Button.led_red
//     Port2 (CANEO series10 Hygienic)/IO-Link Port2_out/LED Effect <-> PlcTask Outputs/MAIN.DISABLE_Button.led_effect
//     Port3 (CANEO series10 Hygienic)/IO-Link Port3_in/Actuation Count <-> PlcTask Inputs/MAIN.RESET_Button.actuation_count
//     Port3 (CANEO series10 Hygienic)/IO-Link Port3_in/Actuation Flag <-> PlcTask Inputs/MAIN.RESET_Button.actuation_flag
//     Port3 (CANEO series10 Hygienic)/IO-Link Port3_in/Actuation Strength <-> PlcTask Inputs/MAIN.RESET_Button.actuation_strength
//     Port3 (CANEO series10 Hygienic)/IO-Link Port3_in/Surrounding Brightness <-> PlcTask Inputs/MAIN.RESET_Button.surrounding_brightness
//     Port3 (CANEO series10 Hygienic)/IO-Link Port3_out/Active LEDs <-> PlcTask Outputs/MAIN.RESET_Button.active_leds
//     Port3 (CANEO series10 Hygienic)/IO-Link Port3_out/Effect Frequency <-> PlcTask Outputs/MAIN.RESET_Button.effect_frequency
//     Port3 (CANEO series10 Hygienic)/IO-Link Port3_out/LED Brightness <-> PlcTask Outputs/MAIN.RESET_Button.led_brightness
//     Port3 (CANEO series10 Hygienic)/IO-Link Port3_out/LED Color B <-> PlcTask Outputs/MAIN.RESET_Button.led_blue
//     Port3 (CANEO series10 Hygienic)/IO-Link Port3_out/LED Color G <-> PlcTask Outputs/MAIN.RESET_Button.led_green
//     Port3 (CANEO series10 Hygienic)/IO-Link Port3_out/LED Color R <-> PlcTask Outputs/MAIN.RESET_Button.led_red
//     Port3 (CANEO series10 Hygienic)/IO-Link Port3_out/LED Effect <-> PlcTask Outputs/MAIN.RESET_Button.led_effect
//   IoLink PushButtons (EP6224-0002) <-> PLC1/PLC1 Instance
//     Port1 (CANEO series10 Hygienic)/IO-Link Port1_in/Actuation Count <-> PlcTask Inputs/MAIN.START_Button.actuation_count
//     Port1 (CANEO series10 Hygienic)/IO-Link Port1_in/Actuation Flag <-> PlcTask Inputs/MAIN.START_Button.actuation_flag
//     Port1 (CANEO series10 Hygienic)/IO-Link Port1_in/Actuation Strength <-> PlcTask Inputs/MAIN.START_Button.actuation_strength
//     Port1 (CANEO series10 Hygienic)/IO-Link Port1_in/Surrounding Brightness <-> PlcTask Inputs/MAIN.START_Button.surrounding_brightness
//     Port1 (CANEO series10 Hygienic)/IO-Link Port1_out/Active LEDs <-> PlcTask Outputs/MAIN.START_Button.active_leds
//     Port1 (CANEO series10 Hygienic)/IO-Link Port1_out/Effect Frequency <-> PlcTask Outputs/MAIN.START_Button.effect_frequency
//     Port1 (CANEO series10 Hygienic)/IO-Link Port1_out/LED Brightness <-> PlcTask Outputs/MAIN.START_Button.led_brightness
//     Port1 (CANEO series10 Hygienic)/IO-Link Port1_out/LED Color B <-> PlcTask Outputs/MAIN.START_Button.led_blue
//     Port1 (CANEO series10 Hygienic)/IO-Link Port1_out/LED Color G <-> PlcTask Outputs/MAIN.START_Button.led_green
//     Port1 (CANEO series10 Hygienic)/IO-Link Port1_out/LED Color R <-> PlcTask Outputs/MAIN.START_Button.led_red
//     Port1 (CANEO series10 Hygienic)/IO-Link Port1_out/LED Effect <-> PlcTask Outputs/MAIN.START_Button.led_effect
//     Port2 (CANEO series10 Hygienic)/IO-Link Port2_in/Actuation Count <-> PlcTask Inputs/MAIN.DISABLE_Button.actuation_count
//     Port2 (CANEO series10 Hygienic)/IO-Link Port2_in/Actuation Flag <-> PlcTask Inputs/MAIN.DISABLE_Button.actuation_flag
//     Port2 (CANEO series10 Hygienic)/IO-Link Port2_in/Actuation Strength <-> PlcTask Inputs/MAIN.DISABLE_Button.actuation_strength
//     Port2 (CANEO series10 Hygienic)/IO-Link Port2_in/Surrounding Brightness <-> PlcTask Inputs/MAIN.DISABLE_Button.surrounding_brightness
//     Port2 (CANEO series10 Hygienic)/IO-Link Port2_out/Active LEDs <-> PlcTask Outputs/MAIN.DISABLE_Button.active_leds
//     Port2 (CANEO series10 Hygienic)/IO-Link Port2_out/Effect Frequency <-> PlcTask Outputs/MAIN.DISABLE_Button.effect_frequency
//     Port2 (CANEO series10 Hygienic)/IO-Link Port2_out/LED Brightness <-> PlcTask Outputs/MAIN.DISABLE_Button.led_brightness
//     Port2 (CANEO series10 Hygienic)/IO-Link Port2_out/LED Color B <-> PlcTask Outputs/MAIN.DISABLE_Button.led_blue
//     Port2 (CANEO series10 Hygienic)/IO-Link Port2_out/LED Color G <-> PlcTask Outputs/MAIN.DISABLE_Button.led_green
//     Port2 (CANEO series10 Hygienic)/IO-Link Port2_out/LED Color R <-> PlcTask Outputs/MAIN.DISABLE_Button.led_red
//     Port2 (CANEO series10 Hygienic)/IO-Link Port2_out/LED Effect <-> PlcTask Outputs/MAIN.DISABLE_Button.led_effect
//     Port3 (CANEO series10 Hygienic)/IO-Link Port3_in/Actuation Count <-> PlcTask Inputs/MAIN.RESET_Button.actuation_count
//     Port3 (CANEO series10 Hygienic)/IO-Link Port3_in/Actuation Flag <-> PlcTask Inputs/MAIN.RESET_Button.actuation_flag
//     Port3 (CANEO series10 Hygienic)/IO-Link Port3_in/Actuation Strength <-> PlcTask Inputs/MAIN.RESET_Button.actuation_strength
//     Port3 (CANEO series10 Hygienic)/IO-Link Port3_in/Surrounding Brightness <-> PlcTask Inputs/MAIN.RESET_Button.surrounding_brightness
//     Port3 (CANEO series10 Hygienic)/IO-Link Port3_out/Active LEDs <-> PlcTask Outputs/MAIN.RESET_Button.active_leds
//     Port3 (CANEO series10 Hygienic)/IO-Link Port3_out/Effect Frequency <-> PlcTask Outputs/MAIN.RESET_Button.effect_frequency
//     Port3 (CANEO series10 Hygienic)/IO-Link Port3_out/LED Brightness <-> PlcTask Outputs/MAIN.RESET_Button.led_brightness
//     Port3 (CANEO series10 Hygienic)/IO-Link Port3_out/LED Color B <-> PlcTask Outputs/MAIN.RESET_Button.led_blue
//     Port3 (CANEO series10 Hygienic)/IO-Link Port3_out/LED Color G <-> PlcTask Outputs/MAIN.RESET_Button.led_green
//     Port3 (CANEO series10 Hygienic)/IO-Link Port3_out/LED Color R <-> PlcTask Outputs/MAIN.RESET_Button.led_red
//     Port3 (CANEO series10 Hygienic)/IO-Link Port3_out/LED Effect <-> PlcTask Outputs/MAIN.RESET_Button.led_effect

CONFIGURATION PLC1
    RESOURCE PLC ON TwinCAT3
        TASK PlcTask(INTERVAL := T#1ms, PRIORITY := 20);
        PROGRAM MAIN WITH PlcTask : MAIN;
    END_RESOURCE
END_CONFIGURATION

// ---- DemoStep/E_DemoStep.TcDUT
{attribute 'qualified_only'}
{attribute 'strict'}
{attribute 'to_string'}
TYPE E_DemoStep :
(
	ManualMode := -1, // "Do nothing" used to interact with MC3 Motion UI
	Init := 0,
	WaitForIO,
	DetectMovers,
	SortMovers,	
	Enabling,
	SquareUpMovers,
	MoveToSeqenceStartPos,
	JoinTrack,
	FigureEight,
	LeaveTrack,
	GoToOpositeCorner,
	FlyBy,
	MoveAroundPerimeter,
	MoveToCenterOfTiles,
	RotateInverse,
	Spin,
	Lift,
	Tilt,
	Disable
) := ManualMode;
END_TYPE

// ---- DUTs/EStop/E_EStop.TcDUT
{attribute 'qualified_only'}
{attribute 'strict'}
{attribute 'to_string'}
TYPE E_EStop :
(
	Activated		:=0,
	Normallyclosed 	:=3

)BYTE;
END_TYPE

// ---- DUTs/EStop/ST_EstopIO.TcDUT
TYPE ST_EstopIO :
STRUCT
	ch1	AT%I* 	:BIT;
	Ch2	AT%I*	:BIT;	
END_STRUCT
END_TYPE

// ---- DUTs/EStop/U_Estop.TcDUT
TYPE U_Estop :
UNION
	Pos	:E_EStop;	
	IO 	:ST_EstopIO;
END_UNION
END_TYPE

// ---- DUTs/E_ButtonColors.TcDUT
{attribute 'qualified_only'}
{attribute 'strict'}
{attribute 'to_string'}
TYPE E_ButtonColors :
(
	red,
	green,
	blue,
	white
);
END_TYPE

// ---- DUTs/E_UsbLicenseDongleSate.TcDUT
{attribute 'qualified_only'}
{attribute 'strict'}
{attribute 'to_string'}
TYPE E_UsbLicenseDongleSate : // for (C9900-L100 License-Key-USB-Stick) > BoxInfo > BoxStateVar
(
	NO_ERROR			:= 16#0000,	// 0x0000 = No error
	NO_ACTUAL_INPUTS	:= 16#0001,	// 0x0001 = No actual inputs
	NOT_FOUND			:= 16#0004	// 0x0004 = Not found
) UINT:=NOT_FOUND; // this will be overwritten by Real Dongle State
END_TYPE

// ---- DUTs/SelectorSwitch/E_SelectorSwitchPos.TcDUT
{attribute 'qualified_only'}
{attribute 'strict'}
{attribute 'to_string'}
TYPE E_SelectorSwitchPos :
(
	Up := 0,
	Left:=1,
	Right:=2
)BYTE;
END_TYPE

// ---- DUTs/SelectorSwitch/ST_SelectorSwitchIO.TcDUT
TYPE ST_SelectorSwitchIO :
STRUCT
	Left	AT%I* :BIT;
	Right	AT%I* :BIT;	
END_STRUCT
END_TYPE

// ---- DUTs/SelectorSwitch/U_SelectorSwitch.TcDUT
TYPE U_SelectorSwitch :
UNION
	IO :ST_SelectorSwitchIO;
	Pos	:E_SelectorSwitchPos;
END_UNION
END_TYPE

// ---- GVLs/CoorPoint2Tile.TcGVL
//{attribute 'qualified_only'}
VAR_GLOBAL CONSTANT
	RIGHT	: LREAL:=180.0;
	CENTER	: LREAL:=120.0;	
	LEFT	: LREAL:=60.0;
	//---
	TOP_UPPER		: LREAL:=420.0;
	TOP_MIDDLE		: LREAL:=360.0;
	TOP_LOWER		: LREAL:=300.0;
	MEDIAN			: LREAL:=240.0;
	BOTTOM_UPPER	: LREAL:=180.0;
	BOTTOM_MIDDLE	: LREAL:=120.0;
	BOTTOM_LOWER	: LREAL:=60.0;
	//---
	TOP_UPPER_RIGHT,TOP_RIGHT			: ST_POINT := (X := RIGHT,	Y := TOP_UPPER);
	TOP_UPPER_CENTER					: ST_POINT := (X := CENTER,	Y := TOP_UPPER);
	TOP_UPPER_LEFT,TOP_LEFT				: ST_POINT := (X := LEFT,	Y := TOP_UPPER);
	TOP_MIDDLE_RIGHT					: ST_POINT := (X := RIGHT,	Y := TOP_MIDDLE);
	TOP_MIDDLE_CENTER,TOP_CENTER		: ST_POINT := (X := CENTER,	Y := TOP_MIDDLE);
	TOP_MIDDLE_LEFT						: ST_POINT := (X := LEFT,	Y := TOP_MIDDLE);
	TOP_LOWER_RIGHT						: ST_POINT := (X := RIGHT,	Y := TOP_LOWER);
	TOP_LOWER_CENTER					: ST_POINT := (X := CENTER,	Y := TOP_LOWER);
	TOP_LOWER_LEFT						: ST_POINT := (X := LEFT,	Y := TOP_LOWER);
	MEDIAN_RIGHT						: ST_POINT := (X := RIGHT,	Y := MEDIAN);
	MEDIAN_CENTER, PRIME_MIDDLE			: ST_POINT := (X := CENTER,	Y := MEDIAN);
	MEDIAN_LEFT							: ST_POINT := (X := LEFT,	Y := MEDIAN);
	BOTTOM_UPPER_RIGHT					: ST_POINT := (X := RIGHT,	Y := BOTTOM_UPPER);
	BOTTOM_UPPER_CENTER					: ST_POINT := (X := CENTER,	Y := BOTTOM_UPPER);	
	BOTTOM_UPPER_LEFT					: ST_POINT := (X := LEFT,	Y := BOTTOM_UPPER);
	BOTTOM_MIDDLE_RIGHT					: ST_POINT := (X := RIGHT,	Y := BOTTOM_MIDDLE);
	BOTTOM_MIDDLE_CENTER,BOTTOM_CENTER	: ST_POINT := (X := CENTER,	Y := BOTTOM_MIDDLE);
	BOTTOM_MIDDLE_LEFT					: ST_POINT := (X := LEFT,	Y := BOTTOM_MIDDLE);
	BOTTOM_LOWER_RIGHT,BOTTOM_RIGHT		: ST_POINT := (X := RIGHT,	Y := BOTTOM_LOWER);
	BOTTOM_LOWER_CENTER					: ST_POINT := (X := CENTER,	Y := BOTTOM_LOWER);
	BOTTOM_LOWER_LEFT,BOTTOM_LEFT		: ST_POINT := (X := LEFT,	Y := BOTTOM_LOWER);
END_VAR
(*
       2-Tile layout of (x,y) ST_Points          
        (positions marked with `*` Asteriks)     
(0,480)                                 (240,480)
       ┌───────────────┐───────────────┐         
       │               │               │         
       │               │               │         
  upper│       *       *       *       │         
       │               │               │         
       │            TOP│               │         
 middle│───────*───────*───────*───────│         
       │               │TILE           │         
       │               │               │         
  lower│       *       *       *       │         
       │               │               │         
       │               │               │         
 median├───────*───────*───────*───────┤        
       │               │               │         
       │               │               │         
  upper│       *       *       *       │         
       │               │               │         
       │         BOTTOM│               │         
 middle│───────*───────*───────*───────│         
       │               │TILE           │         
       │               │               │         
  lower│       *       *       *       │         
       │               │               │         
       │               │               │         
       └───────────────┘───────────────┘         
  (0,0)      left    center   right     (240,0)  
*)

// ---- GVLs/Defaults.TcGVL
//{attribute 'qualified_only'}
VAR_GLOBAL CONSTANT
	//Move dynamics                 	
	DEFAULT_MOVE			: 	ST_MoveDynamics := (Velocity := 500.0, 	Accel := 1000.0,	Decel := 1000.0,	Jerk := 200000.0); 
	DEFAULT_ROTATE			: 	ST_MoveDynamics := (Velocity := 5.0, 	Accel := 20.0, 		Decel := 20.0, 		Jerk := 100.0);  
END_VAR

// ---- DemoStep/I_BothMovers.TcIO
INTERFACE I_BothMovers EXTENDS I_SingleMover

PROPERTY Mover2 : I_XPlanarMover
GET
END_GET
SET
END_SET
END_PROPERTY

END_INTERFACE

// ---- DemoStep/I_Errorable.TcIO
INTERFACE I_Errorable EXTENDS I_Base

PROPERTY Error : BOOL
GET
END_GET
END_PROPERTY

END_INTERFACE

// ---- DemoStep/I_SingleMover.TcIO
INTERFACE I_SingleMover EXTENDS I_Base

PROPERTY Mover1 : I_XPlanarMover
GET
END_GET
SET
END_SET
END_PROPERTY

METHOD SetMovers : BOOL
VAR_INPUT
	M1, M2 : I_XPlanarMover := 0;
END_VAR
END_METHOD

END_INTERFACE

// ---- DemoStep/I_XplanarTable.TcIO
INTERFACE I_XplanarTable EXTENDS I_Base, I_DemoStep

PROPERTY Table : I_XPlanarSystem
GET
END_GET
SET
END_SET
END_PROPERTY

END_INTERFACE

// ---- DemoStep/I_DemoStep.TcIO
INTERFACE I_DemoStep EXTENDS I_Cyclic

METHOD CyclicLogic
END_METHOD

{attribute 'monitoring' := 'call'}
PROPERTY Done : BOOL
GET
END_GET
END_PROPERTY

METHOD Reset : BOOL
VAR_INPUT
END_VAR
END_METHOD

END_INTERFACE

// ---- POUs/I_DemoSystem.TcIO
INTERFACE I_DemoSystem EXTENDS I_Base

END_INTERFACE

// ---- POUs/MAIN.TcPOU
PROGRAM MAIN
VAR
	SimStart AT %I*			: 	BOOL;// These are inputs that are unlinked for writing conveninece
	SimDisable AT %I*		:	BOOL;
	// Initialized for AutoStart when IO is disabled
	//SelectorSwitch: U_SelectorSwitch := (Pos := E_SelectorSwitchPos.Left);
	START_Button : FB_ToggleButton := (button_type := 1);
	DISABLE_Button : FB_ToggleButton  := (button_type := 2);
	RESET_Button : FB_PushButton := (button_type := 3);
	RestartTimer: TON := (PT := TIME#3S0MS);
	// Initialized for AutoStart when IO is disabled
	//Estop					:	U_Estop := (Pos := E_EStop.Normallyclosed);
	Step					:	E_DemoStep:=E_DemoStep.Init;
	
//	XPlanarDemo				:	FB_XPlanar2TileDemo;
	XPlanarTable  			:	FB_Component_XPlanar;
	Mover1		  			:	FB_XPlanarMover;
	Mover2		  			:	FB_XPlanarMover;
	Track1		 			:	FB_XPlanarTrackSegment;	
	
// DEMO STEPS
	dsInit			 : InitStep 			:= (XPlanarSys:=XPlanarTable, MoveDyn:=DEFAULT_MOVE, RotateDyn:=DEFAULT_ROTATE);
	//dsWaitForIO		 : WaitForRotSW			:= (SelectorSwitch:=SelectorSwitch,
	dsWaitForIO		 : WaitForPB			:= (StartPB:=START_Button,
												SimStart:=SimStart, SimDisable:=SimDisable);
	dsDetectMovers	 : DetectXplanarMovers 	:= (XPlanarSys:=XPlanarTable, DesiredNumberOfMovers:=SYSTEM_MOVER_COUNT);
	dsSortMovers	 : SimpleSort2Movers	:= (M1:=Mover1, M2:=Mover2);
	dsSquareUpMovers : SquareUpMovers		:= (M1:=Mover1, M2:=Mover2);
	dsMoveToStartPos : RecoverMoveToAnyPos	:= (M1TargetPos:=START_POS_MOVER1, M2TargetPos:=START_POS_MOVER2);
	dsJoinTrack		 : JoinAllClosestTracks	:= (XPlanarSys:=XPlanarTable);
	dsFigure8Loop	 : SameTrackMove		:= (Track:=Track1, nLaps:=5, M1EndTrackPos:=864.0, M2EndTrackPos:=651.0,
												TrackMoveDynamics := FIGURE_EIGHT_MOVE);
	dsLeaveTrack	 : LeaveAllTracks		:= (M1TargetPos:=BOTTOM_LEFT,M2TargetPos:=TOP_RIGHT);
	dsFlyBy			 : FlyByMove			:= (FlyByMoveDynamics:=FLY_BY_MOVE, Cycles:=4);
	dsPerimeterMove	 : MoveAroundPerimeter	:= (PerimeterMoveDynamics:=PERIMETER_MOVE,numCycles:=2,bClockwise:=FALSE);
	dsMoveToCenters  : MoveToCenters		;
	dsInvRotate		 : OscillateRotateMove	:= (InverseRotateDynamics:=ROTATE_INVERSE_MOVE, numFlipCycles:=6,RotIncrement:=15.0);
	dsSpin		 	 : SpinMove				:= (SpinRotateDynamics:=SPIN_MOVE,numSpins:=30);
	dsLift		 	 : LiftMove				:= (numLiftCycles:=4);
	dsTilt		 	 : TiltMove				:= (bM1Clockwise:=TRUE,bM2Clockwise:=FALSE);
//	dsDisable		 : SimpleDisableWithRotSwAndEstop:=(SelectorSW:=SelectorSwitch,ESTOP:=Estop,
	dsDisable		 : SimpleDisableWithPB	:= (DisablePB:=DISABLE_Button,
												XPlanarSys:=XPlanarTable,M1:=Mover1, M2:=Mover2,Track:=Track1);
	i						: 	UDINT;
	
	MoverStatus				:	ARRAY[1..SYSTEM_MOVER_COUNT] OF CDT_MCTOPLC_PLANAR_MOVER_STD;
	DetectedMoversInfo		: 	XPlanarApplication.ST_TcIoMoverDetectionInfos;
	
	Mover1Target			:	ST_Point;
	Mover2Target			:	ST_Point;
	RotateTarget			:	LREAL;
	Mover1RotateTarget		:	LREAL;
	Mover2RotateTarget		:	LREAL;
	VerticalTarget			:	LREAL;
	FlipFlop				:	BOOL;
	Cycles					:	UINT;
	SubStep					:	UINT;
	
	TwinCATRestart			:	TC_Restart;
	
	rtError					:	R_TRIG;
	rtEstop					: 	R_TRIG;
	
	LicUsbState AT %I* : E_UsbLicenseDongleSate; // license dongle state //UINT;
	IODeviceState AT %I* : UINT;//good is 0;
	XPlanarDeviceState AT %I* : UINT; //good is 0;

END_VAR                      	
VAR CONSTANT
	//Mover Count
	SYSTEM_MOVER_COUNT	    : UDINT := 2;
	                          	
	FIGURE_EIGHT_MOVE		: 	ST_MoveDynamics := (Velocity := 750.0, 	Accel := 5000.0, 	Decel := 5000.0, 	Jerk := 200000.0);               		
	FLY_BY_MOVE				: 	ST_MoveDynamics := (Velocity := 1500.0, Accel := 20000.0, 	Decel := 20000.0, 	Jerk := 200000.0);    
	PERIMETER_MOVE			: 	ST_MoveDynamics := (Velocity := 2000.0, Accel := 20000.0, 	Decel := 20000.0, 	Jerk := 200000.0);
                              	
	ROTATE_INVERSE_MOVE		: 	ST_MoveDynamics := (Velocity := 750.0, 	Accel := 2000.0, 	Decel := 2000.0, 	Jerk := 15000.0);  
	SPIN_MOVE				: 	ST_MoveDynamics := (Velocity := 2500.0, Accel := 4000.0, 	Decel := 4000.0, 	Jerk := 20000.0);
    
	//Move positions                         	
	START_POS_MOVER1		:	ST_Point 	:= 	(X := 60, 		Y := 60);
	START_POS_MOVER2		:	ST_Point 	:= 	(X := 180, 		Y := 180);	
END_VAR

//XplanarDemo.CyclicLogic();
XplanarTable.CyclicLogic();

CASE LicUsbState OF
	E_UsbLicenseDongleSate.NO_ACTUAL_INPUTS,
	E_UsbLicenseDongleSate.NOT_FOUND: 
		RESET_Button.fault_active:=TRUE;
	E_UsbLicenseDongleSate.NO_ERROR: 
		RESET_Button.fault_active:=FALSE;
END_CASE
 

IF XPlanarDeviceState <> 0 THEN
		START_Button.fault_active:=TRUE;
ELSE
		START_Button.fault_active:=FALSE;
END_IF
// Buttons do not do anything yet
START_Button.CyclicLogic(); DISABLE_Button.CyclicLogic(); RESET_Button.CyclicLogic();

CASE Step OF
{region "Init"}	
	E_DemoStep.Init:
		//TODO: Delete vars and set in respective Demo Steps
		dsInit.CyclicLogic();
 		IF dsInit.Done THEN
 			Step := E_DemoStep.WaitForIO; //NEXT STEP
 		END_IF
{endregion}
{region "WaitForSwitch"}
	E_DemoStep.WaitForIO:
		dsWaitForIO.CyclicLogic();
		IF dsWaitForIO.Done THEN
			Step:= E_DemoStep.DetectMovers; //NEXT STEP
		ELSIF dsWaitForIO.Error THEN
			Step:= E_DemoStep.Disable;
		END_IF
		
{endregion}	
{region "DetectMovers"}	
	E_DemoStep.DetectMovers:
		dsDetectMovers.CyclicLogic();
		IF dsDetectMovers.Done THEN
			Step := E_DemoStep.SortMovers; //NEXT STEP
		END_IF	

{endregion}
{region "SortMovers"}	
			
	E_DemoStep.SortMovers:
		dsSortMovers.CyclicLogic();
		IF dsSortMovers.Done THEN
			Step:=E_DemoStep.Enabling; //NEXT STEP
			dsSortMovers.Reset();
		ELSIF dsSortMovers.Error THEN
			//TODO:error handling not all movers passed to inputs
		END_IF	

		
{endregion}	
{region "Enabling"}	

	E_DemoStep.Enabling:
		IF XplanarTable.EnableMovers().Done THEN
			Step:= E_DemoStep.SquareUpMovers; //NEXT STEP
		ELSIF XplanarTable.EnableMovers().Error THEN
			Step:= E_DemoStep.Disable;
		END_IF

	
{endregion}	
{region "DemoStepTemplate"}	
	(*
	E_DemoStep.DemoStepTemplate:	
		
		IF Movers.DoCommand.SquareUp().Done THEN
			Step:= E_DemoStep.NEXT;	//NEXT STEP
		ELSIF Movers.DoCommand().Error THEN
			Step:=E_DemoStep.Disable;
		END_IF
		*)
{endregion}	{region "SquareUpMovers"}	
	
	E_DemoStep.SquareUpMovers:	
		dsSquareUpMovers.CyclicLogic();
		IF dsSquareUpMovers.Done THEN
			Step:=E_DemoStep.MoveToSeqenceStartPos;
			dsSquareUpMovers.Reset();	
		ELSIF dsSortMovers.Error THEN
			Step:=E_DemoStep.Disable;
		END_IF	
		
{endregion}	
{region "MoveToSeqenceStartPos"}
				
	E_DemoStep.MoveToSeqenceStartPos:
		dsMoveToStartPos.CyclicLogic();
		IF dsMoveToStartPos.Done THEN
			Step:=E_DemoStep.JoinTrack;//NEXT STEP
			dsMoveToStartPos.Reset();
		END_IF
		
{endregion}
{region "JoinTrack"}

	E_DemoStep.JoinTrack:
		dsJoinTrack.CyclicLogic();
		IF dsJoinTrack.Done THEN
			Step:=E_DemoStep.FigureEight;//NEXT STEP
			dsJoinTrack.Reset();
		END_IF

{endregion}
{region "FigureEight"}	
	
	E_DemoStep.FigureEight:
			dsFigure8Loop.CyclicLogic();
		IF dsFigure8Loop.Done THEN
			Step:=E_DemoStep.LeaveTrack;//NEXT STEP
			dsFigure8Loop.Reset();
		END_IF
		
{endregion}
{region "LeaveTrack"}	
		
	E_DemoStep.LeaveTrack:
		dsLeaveTrack.CyclicLogic();
		IF dsLeaveTrack.Done THEN
			Step:=E_DemoStep.FlyBy;//NEXT STEP
			dsLeaveTrack.Reset();			
		END_IF	
		
{endregion}
{region "FlyBy"}	
			
	E_DemoStep.FlyBy:		
		dsFlyBy.CyclicLogic();
		IF dsFlyBy.Done THEN
			Step:=E_DemoStep.MoveAroundPerimeter;//NEXT STEP
			dsFlyBy.Reset();			
		END_IF	
		
{endregion}
{region "MoveAroundPerimeter"}	

	E_DemoStep.MoveAroundPerimeter:						
		dsPerimeterMove.CyclicLogic();
		IF dsPerimeterMove.Done THEN
			Step:=E_DemoStep.MoveToCenterOfTiles;//NEXT STEP
			dsPerimeterMove.Reset();			
		END_IF	
		
		
{endregion}	
{region "MoveToCenterOfTiles"}	

	E_DemoStep.MoveToCenterOfTiles:
		dsMoveToCenters.CyclicLogic();
		IF dsMoveToCenters.Done THEN
			Step:=E_DemoStep.RotateInverse;//NEXT STEP
			dsMoveToCenters.Reset();			
		END_IF	
		
{endregion}	
{region "RotateInverse"}	
		
	E_DemoStep.RotateInverse:
		dsInvRotate.CyclicLogic();
		IF dsInvRotate.Done THEN
			Step:=E_DemoStep.Spin;//NEXT STEP
			dsInvRotate.Reset();			
		END_IF
		
{endregion}	
{region "Spin"}
		
	E_DemoStep.Spin:
	dsSpin.CyclicLogic();
		IF dsSpin.Done THEN
			Step:=E_DemoStep.Lift;//NEXT STEP
			dsSpin.Reset();			
		END_IF
	
{endregion}	
{region "Lift"}	

	E_DemoStep.Lift:
	dsLift.CyclicLogic();
		IF dsLift.Done THEN
			Step:=E_DemoStep.Tilt;//NEXT STEP
			dsLift.Reset();			
		END_IF
	
{endregion}	
{region "Tilt"}	
	
	E_DemoStep.Tilt:
		dsTilt.CyclicLogic();
		IF dsTilt.Done THEN
			Step:=E_DemoStep.Init;//NEXT STEP is Init because this is the last step
			dsTilt.Reset();			
		END_IF
				
		
{endregion}			
{region "Disable"}					
    
	E_DemoStep.Disable:
		dsDisable.CyclicLogic();
		IF dsDisable.Done THEN
			Step:=E_DemoStep.Init;//NEXT STEP is Init because this is the last step
			dsDisable.Reset();			
		END_IF
{endregion}			
END_CASE

{region "Error detection"}

	rtError(CLK:=Mover1.Error OR Mover2.Error OR Track1.Error );
	//rtEstop(CLK:=Estop.Pos = E_EStop.Activated );
	IF rtError.Q
	//OR rtEstop.Q THEN
	OR DISABLE_Button.press_event THEN //rising edge of disable button
		Step:=E_DemoStep.Disable;
	END_IF	
	
{endregion}

	
{region "Status update"}

	FOR i:=1 TO XPlanar.MoverCount DO
		IF ip.Movers[i]<>0 THEN		
			MoverStatus[i]:=ip.Movers[i].Status;
		END_IF
	END_FOR
	
{endregion}	


{region "System Restart"}
	//In the event of an unrecovrable error, turn the selector switch to the right
	RestartTimer(IN:= RESET_Button.pressed);
	TwinCATRestart(
		NETID:='' , 
//		RESTART:=SelectorSwitch.Pos = E_SelectorSwitchPos.Right);
		RESTART:=RestartTimer.Q);

{endregion}

END_PROGRAM

// ---- POUs/FB_ToggleButton.TcPOU
FUNCTION_BLOCK FB_ToggleButton
VAR_INPUT
    button_type  : USINT := 0; // 0=other, 1=start, 2=stop, 3=reset
    enabled      : BOOL := TRUE;
    fault_active : BOOL := FALSE;
END_VAR

VAR_OUTPUT
	toggleActive		: BOOL;
    pressed				: BOOL;
    press_event			: BOOL;
    press_count			: UINT;
    touch_strength		: BYTE;
    ambient_brightness	: BYTE;
END_VAR

VAR
    // IO-Link process data inputs
    actuation_flag         AT %I* : BYTE;
    actuation_count        AT %I* : UINT;
    actuation_strength     AT %I* : BYTE;
    surrounding_brightness AT %I* : BYTE;

    // IO-Link process data outputs
    active_leds      AT %Q* : UINT;
    led_brightness   AT %Q* : BYTE;
    led_red          AT %Q* : BYTE;
    led_green        AT %Q* : BYTE;
    led_blue         AT %Q* : BYTE;
    led_effect       AT %Q* : BYTE;
    effect_frequency AT %Q* : BYTE;

    press_edge : R_TRIG;
	_toggle_state : BOOL;
	
	custom_red	: BYTE;
	custom_green: BYTE;
	custom_blue	: BYTE;
	customOn_effect : BYTE:=LED_STATIC;
	customOn_effectFrequency : BYTE:=0;
	customPressed_effect : BYTE:=LED_STATIC;
	customPressed_effectFrequency : BYTE:=0;
//    sH     : STRING := 'AB CD EF 01 23 45 67 89';
//     RGB_DATA   : ARRAY[1..3] OF BYTE;
//     
END_VAR

VAR CONSTANT
    // pushbutton types
    BUTTON_GENERIC : USINT := 0;
    BUTTON_START : USINT := 1;
    BUTTON_STOP  : USINT := 2;
    BUTTON_RESET : USINT := 3;
	BUTTON_CUSTOM : USINT := 5;

    // LED effects
    LED_STATIC : BYTE := 0;
    LED_FLASH  : BYTE := 1;
    LED_PULSE  : BYTE := 2;
END_VAR

CyclicLogic();

PROPERTY Color : E_ButtonColors
SET
CASE Color OF
	E_ButtonColors.red:
		led_red		:= 255;
		led_green	:= 0;
		led_blue	:= 0;
	E_ButtonColors.green:
		led_red		:= 0;
		led_green	:= 255;
		led_blue	:= 0;
	E_ButtonColors.blue:
		led_red		:= 0;
		led_green	:= 0;
		led_blue	:= 255;
	E_ButtonColors.white:
		led_red		:= 255;
		led_green	:= 255;
		led_blue	:= 255;
END_CASE
END_SET
END_PROPERTY

METHOD CyclicLogic : BOOL
VAR_INPUT
END_VAR

// read pushbutton state
	pressed := actuation_flag = 1;
	press_edge(CLK := pressed);
	press_event := press_edge.Q;
	IF press_edge.Q THEN
		_toggle_state:=NOT _toggle_state;
	END_IF
	toggleActive:= _toggle_state;
	press_count := actuation_count;
	touch_strength := actuation_strength;
	ambient_brightness := surrounding_brightness;

// default LED configuration.
THIS^.DefaultLED();	
// disable LED when the pushbutton is disabled
IF NOT enabled THEN
	THIS^.DisableLED();

// fault condition overrides normal behavior
ELSIF fault_active THEN
	//color = red
		led_red := 255;
		led_green := 0;
	    led_blue := 0;
	// effect = flashing fast
		led_brightness := 100;
		led_effect := LED_FLASH;
		effect_frequency := 20;
// normal pushbutton behavior		
ELSE 
	//set brightness
	IF toggleActive THEN //if toggle active
		led_brightness:=80; //on when active
	END_IF
	IF pressed THEN // if button is currently pressed
		led_brightness := 100; //on when pressed
	END_IF
    CASE button_type OF
        BUTTON_START:
			//color = green
				led_red := 0;
				led_green := 255;
				led_blue := 0;
			//effect = off normally, on when pressed
				led_effect := LED_STATIC;
				effect_frequency := 0;
				
        BUTTON_STOP:
            // color = red
				led_red := 255;
				led_green := 0;
				led_blue := 0;
			//effect = off normally, on when pressed
				led_effect := LED_STATIC;
				effect_frequency := 0;
        BUTTON_RESET:
            // color = blue
				led_red := 0;
				led_green := 0;
				led_blue := 255;
			//effect = slow pulse normally, on when pressed
				led_effect := LED_PULSE;
				effect_frequency := 10; // slow pulse makes reset visually distinct
				IF pressed THEN
					led_effect := LED_STATIC;
				END_IF
		BUTTON_GENERIC:
            //color = white
				led_red := 255;
				led_green := 255;
				led_blue := 255;
			//effect = normally off, on when pressed
				led_effect := LED_STATIC;
				effect_frequency := 0;
		ELSE
			// custom button, must set through properties and methods
			            //color = white
				led_red 	:= custom_red; 
				led_green 	:= custom_green;
				led_blue 	:= custom_blue;
			//effect = normally off, on when pressed
				led_effect := customOn_effect;
				effect_frequency :=customOn_effectFrequency;
				IF pressed THEN
					led_effect := customPressed_effect;
					effect_frequency :=customPressed_effectFrequency;
					led_brightness := 100;
				END_IF	
    END_CASE
END_IF
END_METHOD

METHOD DefaultLED : BOOL
VAR_INPUT
END_VAR
active_leds := 1;
led_brightness := 60; //enabled but not active and not pressed
// color = white
	led_red := 255;
	led_green := 255;
	led_blue := 255;
// effect = on
	led_effect := LED_STATIC;
	effect_frequency := 0;
END_METHOD

METHOD DisableLED : BOOL
VAR_INPUT
END_VAR
active_leds := 0;

led_red := 0;
led_green := 0;
led_blue := 0;

led_effect := LED_STATIC;
effect_frequency := 0;
END_METHOD

METHOD setCustomEffect
VAR_INPUT
	On_effect : BYTE:=LED_STATIC;
	On_effectFrequency : BYTE:=0;
	Pressed_effect : BYTE:=LED_STATIC;
	Pressed_effectFrequency : BYTE:=0;
END_VAR
	customOn_effect					:= On_effect; 
	customOn_effectFrequency		:= On_effectFrequency;  
	customPressed_effect			:= Pressed_effect;
	customPressed_effectFrequency	:= Pressed_effectFrequency;
END_METHOD

METHOD setCustomRGB
VAR_INPUT
	red		: BYTE;
    green	: BYTE;
    blue	: BYTE;
END_VAR
custom_red	:= led_red		:= red;  
custom_green:= led_green	:= green;
custom_blue	:= led_blue		:= blue;
END_METHOD

END_FUNCTION_BLOCK

// ---- POUs/FB_PushButton.TcPOU
FUNCTION_BLOCK FB_PushButton
VAR_INPUT
    button_type  : USINT := 0; // 0=other, 1=start, 2=stop, 3=reset
    enabled      : BOOL := TRUE;
    fault_active : BOOL := FALSE;
END_VAR

VAR_OUTPUT
    pressed            : BOOL;
    press_event        : BOOL;
    press_count        : UINT;
    touch_strength     : BYTE;
    ambient_brightness : BYTE;
END_VAR

VAR
    // IO-Link process data inputs
    actuation_flag         AT %I* : BYTE;
    actuation_count        AT %I* : UINT;
    actuation_strength     AT %I* : BYTE;
    surrounding_brightness AT %I* : BYTE;

    // IO-Link process data outputs
    active_leds      AT %Q* : UINT;
    led_brightness   AT %Q* : BYTE;
    led_red          AT %Q* : BYTE;
    led_green        AT %Q* : BYTE;
    led_blue         AT %Q* : BYTE;
    led_effect       AT %Q* : BYTE;
    effect_frequency AT %Q* : BYTE;

    press_edge : R_TRIG;
	_toggle_state : BOOL;
	
	custom_red	: BYTE;
	custom_green: BYTE;
	custom_blue	: BYTE;
	customOn_effect : BYTE:=LED_STATIC;
	customOn_effectFrequency : BYTE:=0;
	customPressed_effect : BYTE:=LED_STATIC;
	customPressed_effectFrequency : BYTE:=0;
//    sH     : STRING := 'AB CD EF 01 23 45 67 89';
//     RGB_DATA   : ARRAY[1..3] OF BYTE;
//     
END_VAR

VAR CONSTANT
    // pushbutton types
    BUTTON_GENERIC : USINT := 0;
    BUTTON_START : USINT := 1;
    BUTTON_STOP  : USINT := 2;
    BUTTON_RESET : USINT := 3;
	BUTTON_CUSTOM : USINT := 5;

    // LED effects
    LED_STATIC : BYTE := 0;
    LED_FLASH  : BYTE := 1;
    LED_PULSE  : BYTE := 2;
END_VAR

CyclicLogic();

PROPERTY Color : E_ButtonColors
SET
CASE Color OF
	E_ButtonColors.red:
		led_red		:= 255;
		led_green	:= 0;
		led_blue	:= 0;
	E_ButtonColors.green:
		led_red		:= 0;
		led_green	:= 255;
		led_blue	:= 0;
	E_ButtonColors.blue:
		led_red		:= 0;
		led_green	:= 0;
		led_blue	:= 255;
	E_ButtonColors.white:
		led_red		:= 255;
		led_green	:= 255;
		led_blue	:= 255;
END_CASE
END_SET
END_PROPERTY

METHOD CyclicLogic : BOOL
VAR_INPUT
END_VAR

// read pushbutton state
	pressed := actuation_flag = 1;
	
	press_edge(CLK := pressed);
	press_event := press_edge.Q;
	
	press_count := actuation_count;
	touch_strength := actuation_strength;
	ambient_brightness := surrounding_brightness;

// default LED configuration.
	active_leds := 1;
	led_brightness := 60;
	// color = white
		led_red := 255;
		led_green := 255;
		led_blue := 255;
	// effect = on
		led_effect := LED_STATIC;
		effect_frequency := 0;

// disable LED when the pushbutton is disabled
IF NOT enabled THEN
    active_leds := 0;
	
    led_red := 0;
    led_green := 0;
    led_blue := 0;
	
    led_effect := LED_STATIC;
    effect_frequency := 0;

// fault condition overrides normal behavior
ELSIF fault_active THEN
	//color = red
		led_red := 255;
		led_green := 0;
	    led_blue := 0;
	// effect = flashing fast
		led_brightness := 100;
		led_effect := LED_FLASH;
		effect_frequency := 20;
// normal pushbutton behavior		
ELSE 
    CASE button_type OF
        BUTTON_START:
			//color = green
				led_red := 0;
				led_green := 255;
				led_blue := 0;
			//effect = off normally, on when pressed
				led_effect := LED_STATIC;
				effect_frequency := 0;
				IF pressed THEN
					led_brightness := 100;
				END_IF
				
        BUTTON_STOP:
            // color = red
				led_red := 255;
				led_green := 0;
				led_blue := 0;
			//effect = off normally, on when pressed
				led_effect := LED_STATIC;
				effect_frequency := 0;
				IF pressed THEN
					led_brightness := 100;
				END_IF
				
        BUTTON_RESET:
            // color = blue
				led_red := 0;
				led_green := 0;
				led_blue := 255;
			//effect = slow pulse normally, on when pressed
				led_effect := LED_PULSE;
				effect_frequency := 10; // slow pulse makes reset visually distinct
				IF pressed THEN
					led_effect := LED_STATIC;
					led_brightness := 100;
				END_IF
		BUTTON_GENERIC:
            //color = white
				led_red := 255;
				led_green := 255;
				led_blue := 255;
			//effect = normally off, on when pressed
				led_effect := LED_STATIC;
				effect_frequency := 0;
				IF pressed THEN
					led_brightness := 100;
				END_IF	
		ELSE
			// custom button, must set through properties and methods
			            //color = white
				led_red 	:= custom_red; 
				led_green 	:= custom_green;
				led_blue 	:= custom_blue;
			//effect = normally off, on when pressed
				led_effect := customOn_effect;
				effect_frequency :=customOn_effectFrequency;
				IF pressed THEN
					led_effect := customPressed_effect;
					effect_frequency :=customPressed_effectFrequency;
					led_brightness := 100;
				END_IF	
    END_CASE
END_IF
END_METHOD

METHOD setCustomEffect
VAR_INPUT
	On_effect : BYTE:=LED_STATIC;
	On_effectFrequency : BYTE:=0;
	Pressed_effect : BYTE:=LED_STATIC;
	Pressed_effectFrequency : BYTE:=0;
END_VAR
	customOn_effect := On_effect; 
	customOn_effectFrequency := On_effectFrequency;  
	customPressed_effect := Pressed_effect;
	customPressed_effectFrequency := Pressed_effectFrequency;
END_METHOD

METHOD setCustomRGB
VAR_INPUT
	red		: BYTE;
    green	: BYTE;
    blue	: BYTE;
END_VAR
custom_red	:= led_red		:= red;  
custom_green:= led_green	:= green;
custom_blue	:= led_blue		:= blue;
END_METHOD

END_FUNCTION_BLOCK

// ---- DemoStep/Steps/InitStep.TcPOU
FUNCTION_BLOCK InitStep IMPLEMENTS I_DemoStep
VAR_INPUT
	XPlanarSys		: 	I_XPlanarSystem;
	MoveDyn			: 	ST_MoveDynamics := (Velocity := 500.0, 	Accel := 1000.0,	Decel := 1000.0,	Jerk := 200000.0); 
	RotateDyn		: 	ST_MoveDynamics := (Velocity := 5.0, 	Accel := 20.0, 		Decel := 20.0, 		Jerk := 100.0);  
END_VAR
VAR_OUTPUT
END_VAR
VAR
	_XPlanarSysInit: I_Initializable;
	_Done			: BOOL;
END_VAR

METHOD CyclicLogic
VAR
END_VAR
// Table Cyclic logic should already be called.
F_SetAllMoversMovement(MoveDyn);
F_SetAllMoversRotation(RotateDyn);

IF XPlanarSys<>0 AND_THEN __QUERYINTERFACE(XPlanarSys, _XPlanarSysInit) THEN
	_Done := _XPlanarSysInit.Initialized;
ELSE 
	_Done:=FALSE;
END_IF
END_METHOD

{attribute 'monitoring' := 'call'}
PROPERTY Done : BOOL
GET
Done:= _Done;
END_GET
END_PROPERTY

METHOD Reset : BOOL
//Not really needed
_Done:=FALSE;
Reset:=TRUE;
END_METHOD

END_FUNCTION_BLOCK

// ---- DemoStep/Steps/WaitForPB.TcPOU
FUNCTION_BLOCK WaitForPB IMPLEMENTS I_DemoStep
VAR_INPUT
	StartPB			: 	REFERENCE TO FB_ToggleButton;// Start Pushbutton for Start/Disable command
	SimStart		: 	REFERENCE TO BOOL;
	SimDisable		: 	REFERENCE TO BOOL;
END_VAR
VAR_OUTPUT
END_VAR
VAR
	//TwinCATRestart : TC_Restart := (NETID:='', RESTART:=FALSE);
	_bDisableInNextStep	: BOOL; // passed to Error Prop
	_Done		: BOOL;
END_VAR

METHOD CyclicLogic
VAR
END_VAR
// Table Cyclic logic should already be called.
_bDisableInNextStep := FALSE;
//E_DemoStep.WaitForSwitch:
IF XPlanar.OperationMode = XPlanarApplication.XPlanarOperationMode.Normal THEN
	//CyclicLogic() called in Main;
		// dont reset done to latch.
	IF StartPB.toggleActive OR StartPB.pressed THEN
		_Done:=TRUE; // E_DemoStep.DetectMovers; //(Usually) 
		//	E_SelectorSwitchPos.Right:	TwinCATRestart(NETID:='', RESTART:=TRUE); // Done in other part of code 
	ELSE
			_bDisableInNextStep:= TRUE; // E_DemoStep.Disable; ==> Error=TRUE
			_Done := FALSE; // OVERWRITE _Done from Start PB.
	END_IF
ELSE // XPlanar TcCOM OperationMode in a Simulation mode
	IF 	SimStart	THEN _Done:= TRUE; END_IF
	IF 	SimDisable 	THEN _bDisableInNextStep:= TRUE; END_IF
END_IF
END_METHOD

{attribute 'monitoring' := 'call'}
PROPERTY Done : BOOL
GET
Done:= _Done;
END_GET
END_PROPERTY

PROPERTY Error : BOOL
GET
Error:= _bDisableInNextStep;
END_GET
END_PROPERTY

METHOD Reset : BOOL
//Not really needed
_bDisableInNextStep := _Done := FALSE;
Reset:=TRUE;
END_METHOD

END_FUNCTION_BLOCK

// ---- DemoStep/Steps/DetectXplanarMovers.TcPOU
FUNCTION_BLOCK DetectXplanarMovers IMPLEMENTS I_DemoStep, I_XplanarTable
VAR_INPUT
	XPlanarSys		: 	I_XPlanarSystem;
	DesiredNumberOfMovers : UDINT := 2 ;
END_VAR
VAR_OUTPUT
END_VAR
VAR
	_DetectedMoversInfo	: 	XPlanarApplication.ST_TcIoMoverDetectionInfos;
	_Done				: BOOL;
	_Reset: BOOL;
END_VAR

METHOD CyclicLogic
//E_DemoStep.DetectMovers:
IF NOT _Reset THEN
	IF XPlanarSys<>0 AND_THEN XPlanarSys.MoverRedetect().Done THEN
		_DetectedMoversInfo		:= XPlanarSys.Utility.GetMoverDetectionInfos();
		_Done := TRUE;
	END_IF	
ELSE
	//skip cycle for reset
END_IF

//might need to wait a cycle to re-trigger 
IF  _DetectedMoversInfo.TotalDetected = DesiredNumberOfMovers THEN //Default to two
	_Done := TRUE;
	_Reset := TRUE;
END_IF
END_METHOD

{attribute 'monitoring' := 'call'}
PROPERTY Done : BOOL
GET
Done:= _Done;
END_GET
END_PROPERTY

METHOD Reset : BOOL
_DetectedMoversInfo.TotalDetected:=0;
_DetectedMoversInfo.TotalExpected:=0;
_Reset:= TRUE;//skip detect cycle
_Done:=FALSE;
END_METHOD

PROPERTY Table : I_XPlanarSystem
GET
Table:=XPlanarSys;
END_GET
SET
XPlanarSys:=Table;
END_SET
END_PROPERTY

PROPERTY TotalMoversDetected : UDINT;
GET
TotalMoversDetected := _DetectedMoversInfo.TotalDetected;
END_GET
END_PROPERTY

END_FUNCTION_BLOCK

// ---- DemoStep/Steps/SimpleSort2Movers.TcPOU
FUNCTION_BLOCK SimpleSort2Movers IMPLEMENTS I_DemoStep, I_BothMovers, I_Errorable
VAR_INPUT
		M1	:	I_XPlanarMover;
		M2	:	I_XPlanarMover;
		SortByY : BOOL := TRUE;
END_VAR
VAR_OUTPUT
END_VAR
VAR
	_Done:BOOL;
	_Error: BOOL;
END_VAR

METHOD CyclicLogic
IF M1<>0 AND_THEN M2<>0 THEN
	_Error:=FALSE;
	IF (SortByY AND_THEN M1.ActualPosition.y < M2.ActualPosition.y)
		OR (NOT SortByY AND_THEN M1.ActualPosition.X < M2.ActualPosition.X) THEN
		ip.Movers[1] 	:= M1;
		ip.Movers[2] 	:= M2;	
	ELSE
		ip.Movers[2] 	:= M1;
		ip.Movers[1] 	:= M2;		
	END_IF	
	_Done:=TRUE;
ELSE
	_Error := TRUE;
END_IF
END_METHOD

{attribute 'monitoring' := 'call'}
PROPERTY Done : BOOL
GET
Done:=_Done;
END_GET
END_PROPERTY

PROPERTY Error : BOOL
GET
Error:= _Error;
END_GET
END_PROPERTY

PROPERTY Mover1 : I_XPlanarMover
GET
IF ip.Movers[1]<>0 THEN
	Mover1:=ip.Movers[1];
ELSE 
	Mover1:=M1;
END_IF
END_GET
SET
IF Mover1<>0 THEN
	ip.Movers[1]:=Mover1;
END_IF
END_SET
END_PROPERTY

PROPERTY Mover2 : I_XPlanarMover
GET
IF ip.Movers[2]<>0 THEN
	Mover2:=ip.Movers[2];
ELSE 
	Mover2:=M2;
END_IF
END_GET
SET
IF Mover2<>0 THEN
	ip.Movers[2]:=Mover2;
END_IF
END_SET
END_PROPERTY

METHOD Reset : BOOL
_Error:=FALSE;
_Done:=FALSE;
Reset:=TRUE;
END_METHOD

METHOD SetMovers : BOOL
VAR_INPUT
	M1	: I_XPlanarMover;
	M2	: I_XPlanarMover;
END_VAR
ip.Movers[1]:=M1;
ip.Movers[2]:=M2;
END_METHOD

END_FUNCTION_BLOCK

// ---- DemoStep/Steps/SquareUpMovers.TcPOU
FUNCTION_BLOCK SquareUpMovers EXTENDS FB_DemoStepBase IMPLEMENTS I_TwoMovers
VAR_INPUT
END_VAR
VAR_OUTPUT
END_VAR
VAR
END_VAR

METHOD CyclicLogic
IF Mover.MoveCommand.SquareUp().Done AND Mover2.MoveCommand.SquareUp().Done THEN
			Done:=TRUE;
ELSIF Mover.MoveCommand.SquareUp().Error OR Mover2.MoveCommand.SquareUp().Error THEN
			Step:=E_DemoStep.Disable;
		END_IF
END_METHOD

{error 'Add property implementation or delete property to use base implementation'}
PROPERTY Done : BOOL
GET
END_GET
END_PROPERTY

{warning 'Add property implementation'}
PROPERTY Mover2 : I_XPlanarMover
GET
END_GET
SET
END_SET
END_PROPERTY

END_FUNCTION_BLOCK

// ---- DemoStep/Steps/RecoverMoveToAnyPos.TcPOU
FUNCTION_BLOCK RecoverMoveToAnyPos IMPLEMENTS I_DemoStep
VAR_INPUT
		M1TargetPos		:	ST_Point 	:= 	BOTTOM_LEFT;
		M2TargetPos		:	ST_Point 	:= 	BOTTOM_UPPER_RIGHT;
END_VAR
VAR_OUTPUT
END_VAR
VAR
	SubStep: USINT;
	M1CurrentPos,M2CurrentPos :	ST_Point;
	M1InterimPos,M2InterimPos :	ST_Point;
	_Done: BOOL;
END_VAR

METHOD CyclicLogic
CASE SubStep OF
	0:	//Save Current Positions
		M1CurrentPos.X:=ip.Movers[1].ActualPosition.x;
		M1CurrentPos.Y:=ip.Movers[1].ActualPosition.y;
		M2CurrentPos.X:=ip.Movers[2].ActualPosition.x;
		M2CurrentPos.Y:=ip.Movers[2].ActualPosition.y;
		//find alignment to decide which is the proper opposing side for Step1
		F_FindCorrectOpposingCornerPosition(
			M1AlignmentPos	:= M1CurrentPos, 
			M2AlignmentPos	:= M2CurrentPos, 
			M1CornerPos		:= M1InterimPos,
			M2CornerPos		:= M2InterimPos);
		SubStep:=1;
	1,4:	//step 1-2: Move laterally to opposing extremes from CURRENT/Initial alignment
			//step 4-5: Move laterally to opposing extremes from TARGET alignment
			IF	ip.Movers[1].MoveCommand.MoveX(M1InterimPos.X).Done AND 
				ip.Movers[2].MoveCommand.MoveX(M2InterimPos.X).Done THEN
				SubStep:=SubStep+1;
			END_IF
	2,5:
		IF	ip.Movers[1].MoveCommand.MoveY(M1InterimPos.Y).Done AND 
			ip.Movers[2].MoveCommand.MoveY(M2InterimPos.Y).Done THEN
			SubStep:=SubStep+1;
		END_IF
	3:	//find alignment to decide which is the proper opposing side for Step3
		F_FindCorrectOpposingCornerPosition(
			M1AlignmentPos	:= M1TargetPos, 
			M2AlignmentPos	:= M2TargetPos, 
			M1CornerPos		:= M1InterimPos,
			M2CornerPos		:= M2InterimPos);
		SubStep:=4;
	6:// step 6: Free move to TARGET positions from proper opposing extremes 
		IF 	ip.Movers[1].MoveCommand.FreeMove(M1TargetPos.X,M1TargetPos.Y).Done AND
			ip.Movers[2].MoveCommand.FreeMove(M2TargetPos.X,M2TargetPos.Y).Done THEN
			_Done	:= TRUE;
			SubStep	:=0;//reset
		END_IF					

END_CASE
END_METHOD

{attribute 'monitoring' := 'call'}
PROPERTY Done : BOOL
GET
Done:=_Done;
END_GET
END_PROPERTY

METHOD Reset : BOOL
_Done:=FALSE;
SubStep:=0;
Reset:=TRUE;
END_METHOD

END_FUNCTION_BLOCK

// ---- POUs/F_FindCorrectOpposingCornerPosition.TcPOU
FUNCTION F_FindCorrectOpposingCornerPosition : BOOL
VAR_INPUT
	M1AlignmentPos : ST_POINT; //from/reference alignment for Mover 1
	M2AlignmentPos : ST_POINT; //from/reference alignment for Mover 2
	M1CornerPos : REFERENCE TO ST_POINT; //to/target corner for Mover 1 ( Method OUTPUT by REFERENCE )
	M2CornerPos : REFERENCE TO ST_POINT; //to/target corner for Mover 2 ( Method OUTPUT by REFERENCE )
END_VAR

//Find a Target Opposing Corner from a respective Position Alignmnet
(*	i.e.	from:	┌──────────┐    to:	┌─────┌────┐ 
					│          │      	│     │ M2 │ 
					│       ▲  │      	│     └────┘ 
					│   ┌───┼┐ │      	│          │ 
					│   │ M2└┼►│      	│          │ 
					│ ┌─┴──┬─┘ │      	│          │ 
					│◄┼┐M1 │   │      	│          │ 
					│ └┼───┘   │      	┌────┐     │ 
					│  ▼       │      	│ M1 │     │ 
					└──────────┘      	└────┴─────┘ 		*)
//find alignment to decide which is the proper opposing side 
IF M1AlignmentPos.Y >= M2AlignmentPos.Y THEN
	//M1 moves to TOP / M2 moves to BOTTOM
	M1CornerPos.Y := TOP_UPPER;
	M2CornerPos.Y := BOTTOM_LOWER;
ELSE
	//M1 moves to BOTTOM / M2 moves to TOP
	M1CornerPos.Y := BOTTOM_LOWER;
	M2CornerPos.Y := TOP_UPPER;
END_IF
IF M1AlignmentPos.X >= M2AlignmentPos.X THEN
	//M1 moves to RIGHT / M2 moves to LEFT
	M1CornerPos.X := RIGHT;
	M2CornerPos.X := LEFT;
ELSE
	//M1 moves to LEFT / M2 moves to RIGHT
	M1CornerPos.X := LEFT;
	M2CornerPos.X := RIGHT;
END_IF

END_FUNCTION

// ---- DemoStep/Steps/JoinAllClosestTracks.TcPOU
FUNCTION_BLOCK JoinAllClosestTracks IMPLEMENTS I_DemoStep, I_XplanarTable
VAR_INPUT
	XPlanarSys		: 	I_XPlanarSystem;
	UseOrientation : BOOL := FALSE;
END_VAR
VAR_OUTPUT
END_VAR
VAR
	_Done				: BOOL;
END_VAR

METHOD CyclicLogic
//E_DemoStep.JoinTrack:
IF XPlanarSys.EnableTracks().Done AND 
	ip.Movers[1].MoveCommand.JoinClosestTrack(UseOrientation).Done AND
	ip.Movers[2].MoveCommand.JoinClosestTrack(UseOrientation).Done 
THEN
	_Done:=TRUE;
END_IF
END_METHOD

{attribute 'monitoring' := 'call'}
PROPERTY Done : BOOL
GET
Done:= _Done;
END_GET
END_PROPERTY

METHOD Reset : BOOL
_Done:=FALSE;
Reset:=TRUE;
END_METHOD

PROPERTY Table : I_XPlanarSystem
GET
Table:=XPlanarSys;
END_GET
SET
XPlanarSys:=Table;
END_SET
END_PROPERTY

END_FUNCTION_BLOCK

// ---- DemoStep/Steps/SameTrackMove.TcPOU
FUNCTION_BLOCK SameTrackMove IMPLEMENTS I_DemoStep
VAR_INPUT
	Track			: I_XPlanarTrack;
	nLaps			: INT := 0;
	M1EndTrackPos	: LREAL;
	M2EndTrackPos	: LREAL;
	Gap				: LREAL:=30.0;
	moveDirection	: XPlanarApplication.MC_DIRECTION := XPlanarApplication.MC_DIRECTION.mcDirectionNonModulo;
	TrackMoveDynamics: ST_MoveDynamics:=Defaults.DEFAULT_MOVE;
END_VAR
VAR_OUTPUT
END_VAR
VAR
	SubStep: USINT;
	_Done: BOOL;
END_VAR

METHOD CyclicLogic
VAR
END_VAR
CASE SubStep OF
	0:	
		F_SetAllMoversMovement(TrackMoveDynamics);// set move dynamics
		SubStep:=1;
	1:
		IF 	ip.Movers[1].MoveCommand.TrackMove(M1EndTrackPos+(nLaps*Track.TrackLength),Gap,Track,moveDirection).Done AND 
		 	ip.Movers[2].MoveCommand.TrackMove(M2EndTrackPos+(nLaps*Track.TrackLength),Gap,Track,moveDirection).Done 
		THEN
			_Done	:= TRUE;
			SubStep	:=0;//reset
		END_IF					

END_CASE
END_METHOD

{attribute 'monitoring' := 'call'}
PROPERTY Done : BOOL
GET
Done:=_Done;
END_GET
END_PROPERTY

METHOD Reset : BOOL
_Done:=FALSE;
SubStep:=0;
Reset:=TRUE;
END_METHOD

END_FUNCTION_BLOCK

// ---- DemoStep/Steps/LeaveAllTracks.TcPOU
FUNCTION_BLOCK LeaveAllTracks IMPLEMENTS I_DemoStep
VAR_INPUT
	M1TargetPos	: ST_POINT;
	M2TargetPos	: ST_POINT;
	UseOrientation : BOOL := FALSE;

END_VAR
VAR_OUTPUT
END_VAR
VAR
	_Done: BOOL;
END_VAR

METHOD CyclicLogic
VAR
END_VAR
IF 	ip.Movers[1].MoveCommand.LeaveTrack(M1TargetPos.X,M1TargetPos.Y,useOrientation).Done AND
	ip.Movers[2].MoveCommand.LeaveTrack(M2TargetPos.X,M2TargetPos.Y,useOrientation).Done 
THEN
	_Done:=TRUE;		
END_IF
END_METHOD

{attribute 'monitoring' := 'call'}
PROPERTY Done : BOOL
GET
Done:=_Done;
END_GET
END_PROPERTY

METHOD Reset : BOOL
_Done:=FALSE;
Reset:=TRUE;
END_METHOD

END_FUNCTION_BLOCK

// ---- DemoStep/Steps/FlyByMove.TcPOU
FUNCTION_BLOCK FlyByMove IMPLEMENTS I_DemoStep
VAR_INPUT
	FlyByMoveDynamics : ST_MoveDynamics:=(Velocity := 1500.0, Accel := 20000.0, 	Decel := 20000.0, 	Jerk := 200000.0);
	Cycles: USINT:=1;
END_VAR
VAR_OUTPUT
END_VAR
VAR
	SubStep: USINT;
	_Done: BOOL;
	_CycleCount: INT;
	_FlipFlop: BOOL;
	//_M1IsOnLeftSide:BOOL;
	M1CurrentPos,M2CurrentPos :	ST_Point;
	Mover1Target: ST_POINT;
	Mover2Target: ST_POINT;
END_VAR

METHOD CyclicLogic
VAR
END_VAR
CASE SubStep OF
	0:	
		F_SetAllMoversMovement(FlyByMoveDynamics);
		_CycleCount		:=0;
		_FlipFlop	:=FALSE;
		//Save Current Positions
		M1CurrentPos.X:=ip.Movers[1].ActualPosition.x;
		M1CurrentPos.Y:=ip.Movers[1].ActualPosition.y;
		M2CurrentPos.X:=ip.Movers[2].ActualPosition.x;
		M2CurrentPos.Y:=ip.Movers[2].ActualPosition.y;
		//find alignment to decide which is the proper opposing side for Step1
		F_FindCorrectOpposingCornerPosition(
			M1AlignmentPos	:= M1CurrentPos, 
			M2AlignmentPos	:= M2CurrentPos, 
			M1CornerPos		:= Mover1Target,
			M2CornerPos		:= Mover2Target);
		SubStep:=1;
	1:	//step 1: Move laterally to nearer edge from CURRENT/Initial alignment
		IF	ip.Movers[1].MoveCommand.MoveX(Mover1Target.X).Done AND 
			ip.Movers[2].MoveCommand.MoveX(Mover2Target.X).Done THEN
			// x / left or right (this step might be redundant due to Fuction call F_FindCorrectOpposingCornerPosition()
			IF ip.Movers[1].ActualPosition.X > ip.Movers[2].ActualPosition.X THEN
				Mover1Target.X:=RIGHT;
				Mover2Target.X:=LEFT;
			ELSE
				Mover1Target.X:=LEFT;
				Mover2Target.X:=RIGHT;
			END_IF			
			SubStep:=2;

		END_IF
	2:
		IF _FlipFlop THEN
			Mover1Target.Y:=TOP_UPPER;
			Mover2Target.Y:=BOTTOM_LOWER;
		ELSE
			Mover1Target.Y:=BOTTOM_LOWER;
			Mover2Target.Y:=TOP_UPPER;				
		END_IF
		
		IF 	ip.Movers[1].MoveCommand.MoveY(Mover1Target.Y).Done AND
			ip.Movers[2].MoveCommand.MoveY(Mover2Target.Y).Done
		THEN
			IF _FlipFlop THEN //Cycle completed
				_CycleCount:=_CycleCount+1;
				IF _CycleCount=Cycles THEN
					_Done			:=TRUE;
					_CycleCount			:=0;
					SubStep			:=0;
				END_IF
			END_IF
			
			_FlipFlop	:=NOT _FlipFlop;
		END_IF

END_CASE
END_METHOD

{attribute 'monitoring' := 'call'}
PROPERTY Done : BOOL
GET
Done:=_Done;
END_GET
END_PROPERTY

METHOD Reset : BOOL
_Done:=FALSE;
SubStep:=0;
Reset:=TRUE;
END_METHOD

END_FUNCTION_BLOCK

// ---- DemoStep/Steps/MoveAroundPerimeter.TcPOU
FUNCTION_BLOCK MoveAroundPerimeter IMPLEMENTS I_DemoStep
VAR_INPUT
	PerimeterMoveDynamics : 	ST_MoveDynamics := (Velocity := 2000.0, Accel := 20000.0, 	Decel := 20000.0, 	Jerk := 200000.0);
	numCycles: USINT:=1;
	bClockwise :BOOL:= FALSE;// CCW by default
END_VAR
VAR_OUTPUT
END_VAR
VAR
	SubStep: USINT;
	_Done: BOOL;
	_CycleCount: INT;
	_CornerCount: INT;
	_CornerStep: USINT;
	M1CurrentPos,M2CurrentPos :	ST_Point;
	Mover1Target: ST_POINT;
	Mover2Target: ST_POINT;
END_VAR

METHOD CyclicLogic
// E_DemoStep.MoveAroundPerimeter:						
	CASE SubStep OF 
		0:
			F_SetAllMoversMovement(PerimeterMoveDynamics);//Save Current Positions
			M1CurrentPos.X:=ip.Movers[1].ActualPosition.x;
			M1CurrentPos.Y:=ip.Movers[1].ActualPosition.y;
			M2CurrentPos.X:=ip.Movers[2].ActualPosition.x;
			M2CurrentPos.Y:=ip.Movers[2].ActualPosition.y;
			//find alignment to decide which is the proper opposing side for Step1
			F_FindCorrectOpposingCornerPosition(
				M1AlignmentPos	:= M1CurrentPos, 
				M2AlignmentPos	:= M2CurrentPos, 
				M1CornerPos		:= Mover1Target,
				M2CornerPos		:= Mover2Target);
			_CornerCount:=0;
			_CornerStep:=0;
			_CycleCount:=0;
			SubStep:=1;
		// Move to a starting corner.
		1:
			IF	ip.Movers[1].MoveCommand.MoveX(Mover1Target.X).Done AND 
				ip.Movers[2].MoveCommand.MoveX(Mover2Target.X).Done THEN
				SubStep:=2;
			END_IF
		2: 
			IF	ip.Movers[1].MoveCommand.MoveY(Mover1Target.Y).Done AND 
				ip.Movers[2].MoveCommand.MoveY(Mover2Target.Y).Done THEN
				SubStep:=3;
				
			END_IF
		3: // cyclic Perimiter moves from any starting corner
			M1CurrentPos:=Mover1Target;
			M2CurrentPos:=Mover2Target;
			IF NextCornerTarget(CornerStep:=_CornerStep) THEN
				subStep := SubStep+1;
				_CornerCount:=_CornerCount+1;
			END_IF
		4:
			IF (Mover1Target.X <> M1CurrentPos.X OR Mover2Target.X <> M2CurrentPos.X) AND (Mover1Target.X <> Mover2Target.X) THEN
				IF	ip.Movers[1].MoveCommand.MoveX(Mover1Target.X).Done AND 
					ip.Movers[2].MoveCommand.MoveX(Mover2Target.X).Done THEN
					SubStep:=3;
				END_IF
			ELSIF (Mover1Target.Y <> M1CurrentPos.Y OR Mover2Target.Y <> M2CurrentPos.Y) AND (Mover1Target.Y <> Mover2Target.Y) THEN
				IF	ip.Movers[1].MoveCommand.MoveY(Mover1Target.Y).Done AND 
					ip.Movers[2].MoveCommand.MoveY(Mover2Target.Y).Done THEN
					SubStep:=3;
				END_IF
			END_IF
			IF SubStep=3 AND_THEN _CornerCount=4 THEN //Move Complete and-then single cycle complete
				_CycleCount :=_CycleCount+1;
				IF numCycles=_CycleCount THEN
					_Done:=TRUE;
					SubStep:=5;
				ELSE
					_CornerCount:=0;
				END_IF
			END_IF
		5://idle
			_Done:=TRUE;
	END_CASE
END_METHOD

{attribute 'monitoring' := 'call'}
PROPERTY Done : BOOL
GET
Done:=_Done;
END_GET
END_PROPERTY

METHOD FlipTargetXs : BOOL
VAR_INPUT
END_VAR
IF Mover1Target.X >= CENTER THEN
	Mover1Target.X:= LEFT;
ELSE 
	Mover1Target.X:= RIGHT;
END_IF

IF Mover2Target.X <= CENTER THEN
	Mover2Target.X:= RIGHT;
ELSE
	Mover2Target.X:= LEFT;
END_IF
END_METHOD

METHOD FlipTargetYs : BOOL
VAR_INPUT
END_VAR
IF Mover1Target.Y >= MEDIAN THEN
	Mover1Target.Y:= BOTTOM_LOWER;
ELSE 
	Mover1Target.Y:= TOP_UPPER;
END_IF

IF Mover2Target.Y <= MEDIAN THEN
	Mover2Target.Y:= TOP_UPPER;
ELSE
	Mover2Target.Y:= BOTTOM_LOWER;
END_IF
END_METHOD

METHOD NextCornerTarget : BOOL
VAR_IN_OUT
	CornerStep:USINT;
END_VAR

VAR
	NextCoordinateFlip: STRING(INT#1);
END_VAR
(*
				┌----◀------┐(Y)			┌----◀------┐(X)	 (4)┌─────┌────┐(3)
// CCW: (M1)=> BL-▶BR-▶TR-▶TL	CW: (M1)=> BL-▶TL-▶TR-▶BR		 [2]│ TL◀─┼▷TR │[1]
coordinate-flip: (X) (Y) (X) 				 (Y) (X) (Y)		 	│  │  └──┼─┘	
// CCW: [M2]=> TR-▷TL-▷BL-▷BR	CW: [M2]=> TR-▷BR-▷BL-▷TL		    │  △     │ │	
				└----◁------┘(Y)			└----◁------┘(X)	    │  │     ▲ │	
i.e. Directions:												    │  ▼     │ │	
						CCW: ↺⥀ ▼▲◀▶ ⮔	(M1)=>(position)		    │  │     ▽ │	
						CW : ↻⥁ △▽◁▷	[M2]=>[position]		    ┌──┼─┐   | │	
																 (1)│ BL◁┼─▶BR │(2)
																 [3]└────┴─────┘[4] *)
IF CornerStep = 0 THEN
	// First Calculate the starting current CornerStep;
	IF		(Mover1Target.X=BOTTOM_LEFT.X	AND Mover1Target.Y=BOTTOM_LEFT.Y) AND_THEN
			(Mover2Target.X=TOP_RIGHT.X		AND	Mover2Target.Y=TOP_RIGHT.Y) THEN
		CornerStep:=1;
	ELSIF	(Mover1Target.X=BOTTOM_RIGHT.X	AND Mover1Target.Y=BOTTOM_RIGHT.Y) AND_THEN
			(Mover2Target.X=TOP_LEFT.X		AND Mover2Target.Y=TOP_LEFT.Y) THEN
		CornerStep:=2;
	ELSIF	(Mover1Target.X=TOP_RIGHT.X		AND Mover1Target.Y=TOP_RIGHT.Y) AND_THEN
			(Mover2Target.X=BOTTOM_LEFT.X	AND Mover2Target.Y=BOTTOM_LEFT.Y) THEN
		CornerStep:=3;				
	ELSIF	(Mover1Target.X=TOP_LEFT.X		AND Mover1Target.Y=TOP_LEFT.Y) AND_THEN
			(Mover2Target.X=BOTTOM_RIGHT.X	AND Mover2Target.Y=BOTTOM_RIGHT.Y) THEN
		CornerStep:=4;
	END_IF
END_IF
NextCornerTarget:=TRUE;
CASE CornerStep OF //calculate next Corner Step
	1,3:
		IF bClockwise THEN
			FlipTargetYs();
		ELSE
			FlipTargetXs();
		END_IF
	2,4:
		IF bClockwise THEN
			FlipTargetXs();
		ELSE
			FlipTargetYs();
		END_IF
	ELSE 
		// CornerStep still = 0 OR other.
		NextCornerTarget:=FALSE;//error 
		RETURN;
END_CASE
IF NextCornerTarget THEN
	IF bClockwise THEN
		CornerStep:=CornerStep-1;
		IF CornerStep<=0THEN
			CornerStep:=4;
		END_IF
	ELSE
		CornerStep:=CornerStep+1;
		IF CornerStep>=5THEN
			CornerStep:=1;
		END_IF
	END_IF 
END_IF
END_METHOD

METHOD Reset : BOOL
_Done:=FALSE;
SubStep:=0;
Reset:=TRUE;
END_METHOD

END_FUNCTION_BLOCK

// ---- DemoStep/Steps/MoveToCenters.TcPOU
FUNCTION_BLOCK MoveToCenters IMPLEMENTS I_DemoStep
VAR_INPUT
END_VAR
VAR_OUTPUT
END_VAR
VAR
	SubStep: USINT;
	M1CurrentPos, M2CurrentPos	: ST_Point;
	M1TargetPos, M2TargetPos	: ST_Point;
	_Done: BOOL;
END_VAR

METHOD CyclicLogic
CASE SubStep OF
	0:	//Save Current Positions
		M1CurrentPos.X:=ip.Movers[1].ActualPosition.x;
		M1CurrentPos.Y:=ip.Movers[1].ActualPosition.y;
		M2CurrentPos.X:=ip.Movers[2].ActualPosition.x;
		M2CurrentPos.Y:=ip.Movers[2].ActualPosition.y;
		//find alignment to decide which is the proper opposing side for Step1
		F_FindOpposingRotationPosition(
			M1AlignmentPos	:= M1CurrentPos, 
			M2AlignmentPos	:= M2CurrentPos, 
			M1CornerPos		:= M1TargetPos,
			M2CornerPos		:= M2TargetPos);
		SubStep:=1;
	1:
		//step 1-2: Move laterally to opposing extremes from CURRENT/to center alignment
		IF	ip.Movers[1].MoveCommand.MoveY(M1TargetPos.Y).Done AND 
			ip.Movers[2].MoveCommand.MoveY(M2TargetPos.Y).Done THEN
			SubStep:=SubStep+1;
		END_IF
	2:
		IF	ip.Movers[1].MoveCommand.MoveX(M1TargetPos.X).Done AND 
			ip.Movers[2].MoveCommand.MoveX(M2TargetPos.X).Done THEN
			_Done	:= TRUE;
			SubStep	:=0;//reset
		END_IF					

END_CASE
END_METHOD

{attribute 'monitoring' := 'call'}
PROPERTY Done : BOOL
GET
Done:=_Done;
END_GET
END_PROPERTY

METHOD Reset : BOOL
_Done:=FALSE;
SubStep:=0;
Reset:=TRUE;
END_METHOD

END_FUNCTION_BLOCK

// ---- POUs/F_FindOpposingRotationPosition.TcPOU
FUNCTION F_FindOpposingRotationPosition : BOOL
VAR_INPUT
	M1AlignmentPos : ST_POINT; //from/reference alignment for Mover 1
	M2AlignmentPos : ST_POINT; //from/reference alignment for Mover 2
	M1CornerPos : REFERENCE TO ST_POINT; //to/target corner for Mover 1 ( Method OUTPUT by REFERENCE )
	M2CornerPos : REFERENCE TO ST_POINT; //to/target corner for Mover 2 ( Method OUTPUT by REFERENCE )
END_VAR

//Find a Target Opposing tile centers from a respective Position Alignmnet
(*	i.e.	from:	┌──────────┐    to:	┌──────────┐ 
					│          │      	│  ┌────┐  │
					│    ▲     │      	│  │ M2 │  │
					│   ┌┼───┐ │      	│  └────┘  │
					│  ◀┼┘M2 │ │      	│          │
					│ ┌─┴──┬─┘ │      	│          │
					│ │ M1┌┼▶  │      	│  ┌────┐  │
					│ └───┼┘   │      	│  │ M1 │  │
					│     ▼    │      	│  └────┘  │ 
					└──────────┘      	└──────────┘ 		*)
//find alignment to decide which is the proper opposing side 
IF M1AlignmentPos.Y >= M2AlignmentPos.Y THEN
	//M1 moves to TOP / M2 moves to BOTTOM
	M1CornerPos.Y := TOP_MIDDLE;
	M2CornerPos.Y := BOTTOM_MIDDLE;
ELSE 	
	//M1 moves to BOTTOM / M2 moves to TOP
	M1CornerPos.Y := BOTTOM_MIDDLE;
	M2CornerPos.Y := TOP_MIDDLE;
END_IF

M1CornerPos.X := CENTER;
M2CornerPos.X := CENTER;

END_FUNCTION

// ---- DemoStep/Steps/OscillateRotateMove.TcPOU
FUNCTION_BLOCK OscillateRotateMove IMPLEMENTS I_DemoStep
VAR_INPUT
	InverseRotateDynamics : ST_MoveDynamics := (Velocity := 750.0, Accel := 2000.0, Decel := 2000.0, Jerk := 15000.0);
	RotIncrement: LREAL := 15;
	numFlipCycles: UINT:=6;
END_VAR
VAR_OUTPUT
END_VAR
VAR
	SubStep: USINT;
	_Done: BOOL;
	_Cycles: UINT;
	_FlipFlop: BOOL;
	_RotateTarget: LREAL;
	_Mover1RotateTarget: LREAL;
	_Mover2RotateTarget: LREAL;
END_VAR

METHOD CyclicLogic

VAR
END_VAR
CASE SubStep OF
	0:	
		F_SetAllMoversRotation(InverseRotateDynamics);
		_Cycles	:=0;
		_FlipFlop:=FALSE;
		_RotateTarget:=0;
		SubStep:=1;
	1:
		IF _FlipFlop THEN
			_Mover1RotateTarget:=_RotateTarget;
			_Mover2RotateTarget:=(360.0-_RotateTarget)*-1;			
		ELSE
			_Mover1RotateTarget:=(360.0-_RotateTarget)*-1;
			_Mover2RotateTarget:=_RotateTarget;
		END_IF
		
		IF 	ip.Movers[1].MoveCommand.Rotate(_Mover1RotateTarget,0).Done AND
			ip.Movers[2].MoveCommand.Rotate(_Mover2RotateTarget,0).Done
		THEN
			IF _FlipFlop THEN
				_Cycles:=_Cycles+1;
				IF _Cycles>=numFlipCycles THEN
					_Done:=TRUE;
					SubStep:=2;
				ELSE
					_RotateTarget:=_RotateTarget+RotIncrement;
				END_IF
			END_IF
			_FlipFlop:=NOT _FlipFlop;	
		END_IF		

	2://idle
		_Done:=TRUE;
END_CASE
END_METHOD

{attribute 'monitoring' := 'call'}
PROPERTY Done : BOOL
GET
Done:=_Done;
END_GET
END_PROPERTY

METHOD Reset : BOOL
_Done:=FALSE;
SubStep:=0;
Reset:=TRUE;
END_METHOD

END_FUNCTION_BLOCK

// ---- DemoStep/Steps/SpinMove.TcPOU
FUNCTION_BLOCK SpinMove IMPLEMENTS I_DemoStep
VAR_INPUT
	SpinRotateDynamics : ST_MoveDynamics := (Velocity := 2500.0, Accel := 4000.0, Decel := 4000.0, Jerk := 20000.0);
	numSpins: DINT := 1;
	finalOrientation: LREAL := 0;
END_VAR
VAR_OUTPUT
END_VAR
VAR
	SubStep: USINT;
	_Done: BOOL;
END_VAR

METHOD CyclicLogic
CASE SubStep OF
	0:	
		F_SetAllMoversRotation(SpinRotateDynamics);
		SubStep:=1;
	1:
		IF 	ip.Movers[1].MoveCommand.Rotate(finalOrientation,(numSpins * -1)).Done AND
			ip.Movers[2].MoveCommand.Rotate(finalOrientation,numSpins).Done
		THEN
			_Done:=TRUE;
		END_IF		

END_CASE
END_METHOD

{attribute 'monitoring' := 'call'}
PROPERTY Done : BOOL
GET
Done:=_Done;
END_GET
END_PROPERTY

METHOD Reset : BOOL
_Done:=FALSE;
SubStep:=0;
Reset:=TRUE;
END_METHOD

END_FUNCTION_BLOCK

// ---- DemoStep/Steps/LiftMove.TcPOU
FUNCTION_BLOCK LiftMove IMPLEMENTS I_DemoStep
VAR_INPUT
	numLiftCycles: UINT:=4;
END_VAR
VAR_OUTPUT
END_VAR
VAR
	SubStep: USINT;
	_Done: BOOL;
	_Cycles: UINT;
	_FlipFlop: BOOL;
	_VerticalTarget: LREAL;
END_VAR

METHOD CyclicLogic
CASE SubStep OF
	0:	
		_Cycles	:=0;
		_FlipFlop:=FALSE;
		SubStep:=1;
	1:
		
		IF _FlipFlop THEN
			_VerticalTarget:=2.0;
		ELSE
			_VerticalTarget:=5.0;
		END_IF
		IF 	ip.Movers[1].MoveCommand.VerticalMove(_VerticalTarget).Done AND
			ip.Movers[2].MoveCommand.VerticalMove(_VerticalTarget).Done
		THEN
			IF _FlipFlop THEN
				_Cycles	:=_Cycles+1;
				IF _Cycles>=numLiftCycles THEN
					_Done:=TRUE;
					SubStep:=2;
				END_IF
			END_IF
			
			_FlipFlop:=NOT _FlipFlop;
		END_IF	
	2://idle
		_Done:=TRUE;
END_CASE
END_METHOD

{attribute 'monitoring' := 'call'}
PROPERTY Done : BOOL
GET
Done:=_Done;
END_GET
END_PROPERTY

METHOD Reset : BOOL
_Done:=FALSE;
SubStep:=0;
Reset:=TRUE;
END_METHOD

END_FUNCTION_BLOCK

// ---- DemoStep/Steps/TiltMove.TcPOU
FUNCTION_BLOCK TiltMove IMPLEMENTS I_DemoStep
VAR_INPUT
	bM1Clockwise : BOOL:=TRUE;
	bM2Clockwise : BOOL:=FALSE;
END_VAR
VAR_OUTPUT
END_VAR
VAR
	SubStep: USINT;
	_Done: BOOL;
	_M1Direction: INT(-1..1);
	_M2Direction: INT(-1..1);
END_VAR

METHOD CyclicLogic
VAR
END_VAR
CASE SubStep OF
	0:
		IF bM1Clockwise THEN
			_M1Direction:=-1;
		ELSE
			_M1Direction:= +1;
		END_IF
		IF bM2Clockwise THEN
			_M2Direction:=-1;
		ELSE
			_M2Direction:= +1;
		END_IF
		
		IF 	ip.Movers[1].MoveCommand.VerticalMove(5).Done AND	ip.Movers[2].MoveCommand.VerticalMove(5).Done
		THEN SubStep:=1; END_IF
	1:
		IF 	ip.Movers[1].MoveCommand.TiltA(2*_M1Direction).Done AND			ip.Movers[2].MoveCommand.TiltA(-2*_M2Direction).Done
		THEN SubStep:=2; END_IF	
	2:
	
		IF 	ip.Movers[1].MoveCommand.TiltA(-2*_M1Direction).Done AND			ip.Movers[2].MoveCommand.TiltA(2*_M2Direction).Done AND
			ip.Movers[1].MoveCommand.TiltB(2*_M1Direction).Done AND			ip.Movers[2].MoveCommand.TiltB(-2*_M2Direction).Done
		THEN SubStep:=3; END_IF
	3:	
		IF 	ip.Movers[1].MoveCommand.TiltB(-2*_M1Direction).Done AND			ip.Movers[2].MoveCommand.TiltB(2*_M2Direction).Done
		THEN SubStep:=4; END_IF	
		
	4:
		IF 	ip.Movers[1].MoveCommand.TiltA(0).Done AND			ip.Movers[2].MoveCommand.TiltA(0).Done
		THEN SubStep:=5; END_IF	
	
	5:
		IF 	ip.Movers[1].MoveCommand.TiltB(0).Done AND			ip.Movers[2].MoveCommand.TiltB(0).Done
		THEN SubStep:=6; END_IF
	
	6:
		IF 	ip.Movers[1].MoveCommand.VerticalMove(2).Done AND	ip.Movers[2].MoveCommand.VerticalMove(2).Done
		THEN _Done:=TRUE; END_IF					
		
END_CASE
END_METHOD

{attribute 'monitoring' := 'call'}
PROPERTY Done : BOOL
GET
Done:=_Done;
END_GET
END_PROPERTY

METHOD Reset : BOOL
_Done:=FALSE;
SubStep:=0;
Reset:=TRUE;
END_METHOD

END_FUNCTION_BLOCK

// ---- DemoStep/Steps/SimpleDisableWithPB.TcPOU
FUNCTION_BLOCK SimpleDisableWithPB IMPLEMENTS I_DemoStep
VAR_INPUT
	XPlanarSys	: I_XPlanarSystem;
	M1			: I_XPlanarMover;
	M2			: I_XPlanarMover;
	Track		: I_XPlanarTrack;
	
	DisablePB	: REFERENCE TO FB_ToggleButton; // toggle active not used
END_VAR
VAR_OUTPUT
END_VAR
VAR
	SubStep: USINT;
	_Done: BOOL;
END_VAR

METHOD CyclicLogic
VAR
END_VAR
IF XPlanarSys<>0 AND M1<>0 AND M2<>0 THEN
		//Wait till the mover has completed is current move. Then disable it.
		//That way operator intervention is prevented to re-align the movers, and mover gracefully stops
	IF NOT M1.Status.Busy.busyMover AND NOT M2.Status.Busy.busyMover THEN
		XPlanarSys.DisableMovers();
	END_IF
	_Done:= FALSE;
	IF 	M1.Status.State		= MC_PLANAR_STATE.Disabled 
		AND M2.Status.State	= MC_PLANAR_STATE.Disabled 
		AND ((__ISVALIDREF(DisablePB) AND_THEN not DisablePB.toggleActive)
		OR XPlanar.OperationMode = XPlanarApplication.XPlanarOperationMode.BasicSimulation)
	THEN
		_Done:= TRUE;
	END_IF
	IF M1.Error THEN
		M1.Reset();
	END_IF

	IF M2.Error THEN
		M2.Reset();
	END_IF
END_IF

IF Track<>0 AND_THEN Track.Error THEN
	Track.Reset();
END_IF
END_METHOD

{attribute 'monitoring' := 'call'}
PROPERTY Done : BOOL
GET
Done:=_Done;
END_GET
END_PROPERTY

METHOD Reset : BOOL
_Done:=FALSE;
SubStep:=0;
Reset:=TRUE;
END_METHOD

END_FUNCTION_BLOCK

// ---- DemoStep/Steps/SimpleDisableWithRotSwAndEstop.TcPOU
FUNCTION_BLOCK SimpleDisableWithRotSwAndEstop IMPLEMENTS I_DemoStep
VAR_INPUT
	XPlanarSys	: I_XPlanarSystem;
	M1			: I_XPlanarMover;
	M2			: I_XPlanarMover;
	Track		: I_XPlanarTrack;
	
	SelectorSW	: REFERENCE TO U_SelectorSwitch;
	ESTOP		: REFERENCE TO U_Estop;
END_VAR
VAR_OUTPUT
END_VAR
VAR
	SubStep: USINT;
	_Done: BOOL;
END_VAR

METHOD CyclicLogic
VAR
END_VAR
IF XPlanarSys<>0 AND M1<>0 AND M2<>0 THEN
		//Wait till the mover has completed is current move. Then disable it.
		//That way operator intervention is prevented to re-align the movers, and mover gracefully stops
	IF NOT M1.Status.Busy.busyMover AND NOT M2.Status.Busy.busyMover THEN
		XPlanarSys.DisableMovers();
	END_IF
	_Done:= FALSE;
	IF 	M1.Status.State		= MC_PLANAR_STATE.Disabled 
		AND M2.Status.State	= MC_PLANAR_STATE.Disabled 
		AND (
			( (__ISVALIDREF(SelectorSW) AND __ISVALIDREF(ESTOP) )
				AND_THEN(SelectorSW.Pos = E_SelectorSwitchPos.Left AND Estop.Pos = E_EStop.Normallyclosed) )
		OR XPlanar.OperationMode = XPlanarApplication.XPlanarOperationMode.BasicSimulation)
	THEN
		_Done:= TRUE;
	END_IF
	IF M1.Error THEN
		M1.Reset();
	END_IF

	IF M2.Error THEN
		M2.Reset();
	END_IF
END_IF

IF Track<>0 AND_THEN Track.Error THEN
	Track.Reset();
END_IF
END_METHOD

{attribute 'monitoring' := 'call'}
PROPERTY Done : BOOL
GET
Done:=_Done;
END_GET
END_PROPERTY

METHOD Reset : BOOL
_Done:=FALSE;
SubStep:=0;
Reset:=TRUE;
END_METHOD

END_FUNCTION_BLOCK

// ---- DemoStep/Steps/MoveAroundInSequence.TcPOU
FUNCTION_BLOCK MoveAroundInSequence IMPLEMENTS I_DemoStep
VAR_INPUT
	PerimeterMoveDynamics : 	ST_MoveDynamics := (Velocity := 2000.0, Accel := 20000.0, 	Decel := 20000.0, 	Jerk := 200000.0);
	Cycles: USINT:=1;
END_VAR
VAR_OUTPUT
	
END_VAR
VAR
	SubStep: USINT;
	_Done: BOOL;
	_CycleCount: INT;
	_FlipFlop: BOOL;
	_M1IsOnLeftSide:BOOL;
	M1CurrentPos,M2CurrentPos :	ST_Point;
	Mover1Target: ST_POINT;
	Mover2Target: ST_POINT;
END_VAR

METHOD CyclicLogic
VAR
END_VAR
// E_DemoStep.MoveAroundPerimeter:						
	CASE SubStep OF 
		0:
			F_SetAllMoversMovement(PerimeterMoveDynamics);//Save Current Positions
		M1CurrentPos.X:=ip.Movers[1].ActualPosition.x;
		M1CurrentPos.Y:=ip.Movers[1].ActualPosition.y;
		M2CurrentPos.X:=ip.Movers[2].ActualPosition.x;
		M2CurrentPos.Y:=ip.Movers[2].ActualPosition.y;
		//find alignment to decide which is the proper opposing side for Step1
		F_FindCorrectOpposingCornerPosition(
			M1AlignmentPos	:= M1CurrentPos, 
			M2AlignmentPos	:= M2CurrentPos, 
			M1CornerPos		:= Mover1Target,
			M2CornerPos		:= Mover2Target);
		SubStep:=1;
		1:
			IF	ip.Movers[1].MoveCommand.MoveX(Mover1Target.X).Done AND 
				ip.Movers[2].MoveCommand.MoveX(Mover2Target.X).Done THEN
				SubStep:=2;
			END_IF
		2: 
			IF	ip.Movers[1].MoveCommand.MoveY(Mover1Target.Y).Done AND 
				ip.Movers[2].MoveCommand.MoveY(Mover2Target.Y).Done THEN
				SubStep:=3;
			END_IF
		3:
		// [M1]=> BL->BR->TR->TL
		// [M2]=> TR->TL->BL->BR
			Mover1Target:=BOTTOM_LEFT;
			Mover2Target:=TOP_RIGHT;
		
		1:
			Mover1Target:=BOTTOM_RIGHT;
			Mover2Target:=TOP_LEFT;
		
		2:
			Mover1Target:=TOP_RIGHT;
			Mover2Target:=BOTTOM_LEFT;	
	
		3:
			Mover1Target:=TOP_LEFT;
			Mover2Target:=BOTTOM_RIGHT;
	END_CASE

	IF 	ip.Movers[1].MoveCommand.FreeMove(Mover1Target.x,Mover1Target.Y).Done AND
		ip.Movers[2].MoveCommand.FreeMove(Mover2Target.x,Mover2Target.Y).Done
	THEN
		IF SubStep=3 THEN //Cycle completed
			Cycles			:=Cycles+1;
			IF Cycles=2 THEN
				_Done:=TRUE;
			ELSE
				SubStep	:=0;
			END_IF
		ELSE
			SubStep	:=SubStep+1;
		END_IF
			
	END_IF
END_METHOD

{attribute 'monitoring' := 'call'}
PROPERTY Done : BOOL
GET
Done:=_Done;
END_GET
END_PROPERTY

METHOD NextCorner : BOOL
VAR_INPUT
	CornerStep:USINT:=0;
	bClockwise: BOOL:=FALSE; // CCW by default
END_VAR

VAR
	NextCoordinateFlip: STRING(INT#1);
END_VAR
	(*
					┌----◀------┐(Y)			┌----◀------┐(X)	 (4)┌─────┌────┐(3)
	// CCW: (M1)=> BL-▶BR-▶TR-▶TL	CW: (M1)=> BL-▶TL-▶TR-▶BR		 [2]│ TL◀─┼▷TR │[1]
	coordinate-flip: (X) (Y) (X) 				 (Y) (X) (Y)		 	│  │  └──┼─┘	
	// CCW: [M2]=> TR-▷TL-▷BL-▷BR	CW: [M2]=> TR-▷BR-▷BL-▷TL		    │  △     │ │	
					└----◁------┘(Y)			└----◁------┘(X)	    │  │     ▲ │	
	i.e. Directions:												    │  ▼     │ │	
							CCW: ↺⥀ ▼▲◀▶ ⮔	(M1)=>(position)		    │  │     ▽ │	
							CW : ↻⥁ △▽◁▷	[M2]=>[position]		    ┌──┼─┐   | │	
																	 (1)│ BL◁┼─▶BR │(2)
																	 [3]└────┴─────┘[4] *)
NextCorner:=FALSE;
IF CornerStep = 0 THEN
	// First Calculate the starting current CornerStep;
	IF		(Mover1Target.X=BOTTOM_LEFT.X	AND Mover1Target.Y=BOTTOM_LEFT.Y) AND_THEN
			(Mover2Target.X=TOP_RIGHT.X		AND	Mover2Target.Y=TOP_RIGHT.Y) THEN
		CornerStep:=1;
	ELSIF	(Mover1Target.X=BOTTOM_RIGHT.X	AND Mover1Target.Y=BOTTOM_RIGHT.Y) AND_THEN
			(Mover2Target.X=TOP_LEFT.X		AND Mover2Target.Y=TOP_LEFT.Y) THEN
		CornerStep:=2;
	ELSIF	(Mover1Target.X=TOP_RIGHT.X		AND Mover1Target.Y=TOP_RIGHT.Y) AND_THEN
			(Mover2Target.X=BOTTOM_LEFT.X	AND Mover2Target.Y=BOTTOM_LEFT.Y) THEN
		CornerStep:=3;				
	ELSIF	(Mover1Target.X=TOP_LEFT.X		AND Mover1Target.Y=TOP_LEFT.Y) AND_THEN
			(Mover2Target.X=BOTTOM_RIGHT.X	AND Mover2Target.Y=BOTTOM_RIGHT.Y) THEN
		CornerStep:=4;
	ELSE 
		//error
		NextCorner:=FALSE;
		RETURN;
	END_IF
END_IF

IF CornerStep <> 0 THEN
	IF bClockwise THEN
		CornerStep:=CornerStep-1;
		IF CornerStep<1 THEN
			CornerStep:=4;
		END_IF
	ELSE // CCW
		CornerStep:=CornerStep+1;
		IF CornerStep>4 THEN
			CornerStep:=1;
		END_IF
	END_IF

	NextCorner:=TRUE;
	CASE CornerStep OF
		1:	Mover1Target:=BOTTOM_LEFT;	Mover2Target:=TOP_RIGHT;
		2:	Mover1Target:=BOTTOM_RIGHT;	Mover2Target:=TOP_LEFT;
		3:	Mover1Target:=TOP_RIGHT;	Mover2Target:=BOTTOM_LEFT;	
		4:	Mover1Target:=TOP_LEFT;		Mover2Target:=BOTTOM_RIGHT;
	END_CASE
	CASE CornerStep OF
		1,3:
			IF bClockwise THEN
				NextCoordinateFlip := 'Y';
			ELSE
				NextCoordinateFlip := 'X';
			END_IF
		2,4:
			IF bClockwise THEN
				NextCoordinateFlip := 'X';
			ELSE
				NextCoordinateFlip := 'Y';
			END_IF
		ELSE
			//error
			NextCorner:=FALSE;
			return;
	END_CASE
END_METHOD

METHOD Reset : BOOL
_Done:=FALSE;
SubStep:=0;
Reset:=TRUE;
END_METHOD

END_FUNCTION_BLOCK

// ---- DemoStep/Steps/WaitForRotSw.TcPOU
FUNCTION_BLOCK WaitForRotSw IMPLEMENTS I_DemoStep
VAR_INPUT
	SelectorSwitch	: 	REFERENCE TO U_SelectorSwitch;
	SimStart		: 	REFERENCE TO BOOL;
	SimDisable		: 	REFERENCE TO BOOL;
END_VAR
VAR_OUTPUT
END_VAR
VAR
	//TwinCATRestart : TC_Restart := (NETID:='', RESTART:=FALSE);
	_bDisableInNextStep	: BOOL; // passed to Error Prop
	_Done		: BOOL;
END_VAR

METHOD CyclicLogic
VAR
END_VAR
// Table Cyclic logic should already be called.
_bDisableInNextStep := _Done := FALSE;
//E_DemoStep.WaitForSwitch:
IF XPlanar.OperationMode = XPlanarApplication.XPlanarOperationMode.Normal THEN
	CASE SelectorSwitch.Pos OF
		E_SelectorSwitchPos.Left:	_Done:= TRUE; // E_DemoStep.DetectMovers; //(Usually) 
		E_SelectorSwitchPos.Up:		_bDisableInNextStep:= TRUE; // E_DemoStep.Disable; ==> Error=TRUE
	//	E_SelectorSwitchPos.Right:	TwinCATRestart(NETID:='', RESTART:=TRUE); // Done in other part of code 
	END_CASE
ELSE // XPlanar TcCOM OperationMode in a Simulation mode
	IF 	SimStart	THEN _Done:= TRUE; END_IF
	IF 	SimDisable 	THEN _bDisableInNextStep:= TRUE; END_IF
END_IF
END_METHOD

{attribute 'monitoring' := 'call'}
PROPERTY Done : BOOL
GET
Done:= _Done;
END_GET
END_PROPERTY

PROPERTY Error : BOOL
GET
Error:= _bDisableInNextStep;
END_GET
END_PROPERTY

METHOD Reset : BOOL
//Not really needed
_bDisableInNextStep := _Done := FALSE;
Reset:=TRUE;
END_METHOD

END_FUNCTION_BLOCK
